KUKA KRL program: ps_601s1.src, ps_601s1.dat

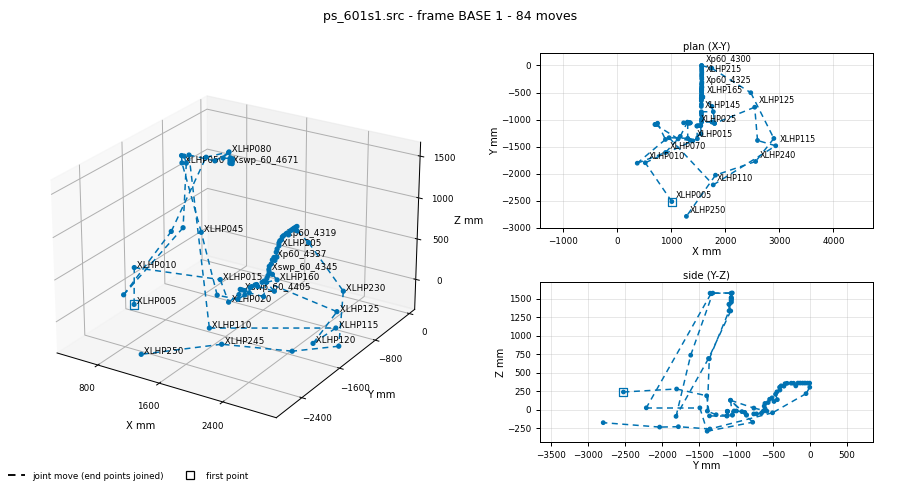
[picture p0: tool path of ps_601s1.src in frame BASE 1, 84 of 89 moves have a stored position in this frame; points joined in program order, loops and branches not executed]
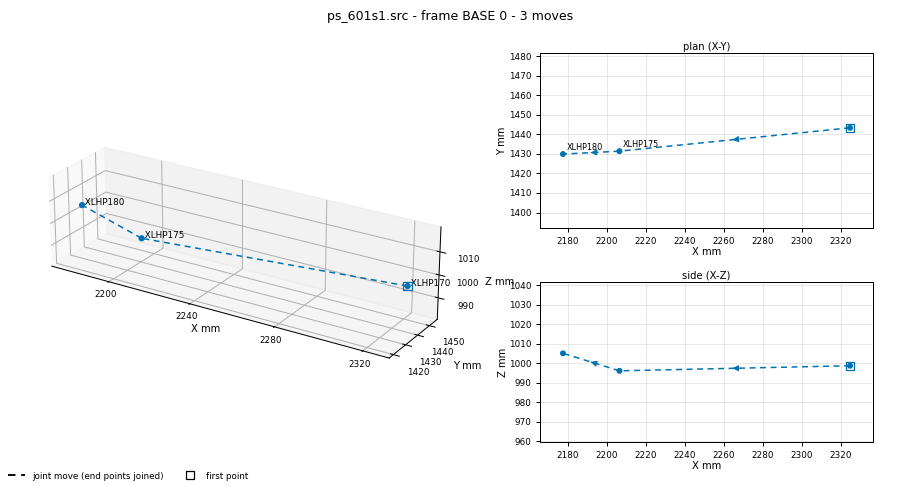
[picture p1: tool path of ps_601s1.src in frame BASE 0, 3 of 89 moves have a stored position in this frame; points joined in program order, loops and branches not executed]
--- ps_601s1.src ---
&ACCESS RVO2
&REL 23
&COMMENT Solda Respot C1 STB
DEF ps_601s1( )
EXT e_Fraes_1()
EXT f_Fraes_1()
;FOLD INI
   ;FOLD BASISTECH INI
      GLOBAL INTERRUPT DECL 3 WHEN $STOPMESS==TRUE DO IR_STOPM ( )
      INTERRUPT ON 3
      BAS (#INITMOV,0 )
   ;ENDFOLD (BASISTECH INI)
   ;FOLD SPOTTECH INI
      USERSPOT(#INIT)
   ;ENDFOLD (SPOTTECH INI)
   ;FOLD GRIPPERTECH INI
      USER_GRP(0,DUMMY,DUMMY,GDEFAULT)
   ;ENDFOLD (GRIPPERTECH INI)
   ;FOLD USER INI
      ;Make your modifications here

   ;ENDFOLD (USER INI)
;ENDFOLD (INI)

; Estacao P13.060 - Robo R1
; Programa: Solda Respot C1 (STB)
; Caracterização dos meios de produção:
; 02/09/2014 09:15 Changes by KUKA Roboter do Brasil

chk_w1_wechs_ok ( )           ; CHECK FERRAMENTA: C1

;FOLD PTP HOME  Vel= 70 % DEFAULT;%{PE}%R 4.1.16,%MKUKATPBASIS,%CMOVE,%VPTP,%P 1:PTP, 2:HOME, 3:, 5:70, 7:DEFAULT
$BWDSTART = FALSE
PDAT_ACT=PDEFAULT
BAS(#PTP_DAT)
FDAT_ACT=FHOME
BAS(#FRAMES)
BAS(#VEL_PTP,70)
$H_POS=XHOME
PTP XHOME
;ENDFOLD

IF (NOT(GHOST())) THEN
IF MaxStandMenge (1) THEN
  MaxStandmengeErreicht (1)
ENDIF

IF Elektrodenwechsel (1) THEN
  e_Fraes_1()
ENDIF
ENDIF

;FOLD OUT 3364 'R1_Solicita Lib. Soldar Geo2' State=TRUE ;%{PE}%R 8.2.20,%MKUKATPBASIS,%COUT,%VOUTX,%P 2:3364, 3:R1_Solicita Lib. Soldar Geo2, 5:TRUE, 6:
$OUT[3364]=TRUE
;ENDFOLD
;FOLD WAIT FOR ( IN 3334 'R1_Aguarda Lib. Soldar Respot' );%{PE}%R 8.2.20,%MKUKATPBASIS,%CEXT_WAIT_FOR,%VEXT_WAIT_FOR,%P 2:, 4:, 5:$IN, 6:3334, 7:R1_Aguarda Lib. Soldar Respot, 9:
WAIT FOR  ( $IN[3334] )
;ENDFOLD
;FOLD OUT 3364 'R1_Solicita Lib. Soldar Geo2' State=FALSE ;%{PE}%R 8.2.20,%MKUKATPBASIS,%COUT,%VOUTX,%P 2:3364, 3:R1_Solicita Lib. Soldar Geo2, 5:FALSE, 6:
$OUT[3364]=FALSE
;ENDFOLD

;FOLD PTP LHP005 CONT Vel=70 % P_OLP1 Tool[1] Base[1];%{PE}%R 4.1.15,%MKUKATPBASIS,%CMOVE,%VPTP,%P 1:PTP, 2:LHP005, 3:C_PTP, 5:70, 7:P_OLP1
$BWDSTART=FALSE
PDAT_ACT=PP_OLP1
BAS (#PTP_DAT )
FDAT_ACT=FLHP005
BAS (#FRAMES )
BAS (#VEL_PTP,70 )
PTP  XLHP005 C_PTP
;ENDFOLD
;FOLD PTP LHP010 CONT Vel= 70 % P_OLP2 Tool[1]:GUN C1 Base[1]:Actros ;%{PE}%R 4.1.16,%MKUKATPBASIS,%CMOVE,%VPTP,%P 1:PTP, 2:LHP010, 3:C_PTP, 5:70, 7:P_OLP2
$BWDSTART = FALSE
PDAT_ACT=PP_OLP2
BAS(#PTP_DAT)
FDAT_ACT=FLHP010
BAS(#FRAMES)
BAS(#VEL_PTP,70)
PTP XLHP010 C_PTP
;ENDFOLD
;FOLD PTP LHP015 CONT Vel= 60 % P_OLP3 Tool[1]:GUN C1 Base[1]:Actros ;%{PE}%R 4.1.16,%MKUKATPBASIS,%CMOVE,%VPTP,%P 1:PTP, 2:LHP015, 3:C_PTP, 5:60, 7:P_OLP3
$BWDSTART = FALSE
PDAT_ACT=PP_OLP3
BAS(#PTP_DAT)
FDAT_ACT=FLHP015
BAS(#FRAMES)
BAS(#VEL_PTP,60)
PTP XLHP015 C_PTP
;ENDFOLD
;FOLD PTP LHP020 CONT Vel= 50 % P_OLP4 Tool[1]:GUN C1 Base[1]:Actros ;%{PE}%R 4.1.16,%MKUKATPBASIS,%CMOVE,%VPTP,%P 1:PTP, 2:LHP020, 3:C_PTP, 5:50, 7:P_OLP4
$BWDSTART = FALSE
PDAT_ACT=PP_OLP4
BAS(#PTP_DAT)
FDAT_ACT=FLHP020
BAS(#FRAMES)
BAS(#VEL_PTP,50)
PTP XLHP020 C_PTP
;ENDFOLD

;FOLD OUT 3331 'R1_Soldando' State=TRUE ;%{PE}%R 8.2.20,%MKUKATPBASIS,%COUT,%VOUTX,%P 2:3331, 3:R1_Soldando, 5:TRUE, 6:
$OUT[3331]=TRUE
;ENDFOLD
;FOLD OUT 3369 'Area de Solda' State=FALSE ;%{PE}%R 8.2.20,%MKUKATPBASIS,%COUT,%VOUTX,%P 2:3369, 3:Area de Solda, 5:FALSE, 6:
$OUT[3369]=FALSE
;ENDFOLD

; Retract Close
;FOLD PTP LHP025 PDAT1 RETR CLS Gun= 1 Tool[1]:GUN C1 Base[1]:Actros ;%{PE}%R 4.1.12,%MKUKATPSPOT,%CRETR,%VPTP,%P 1:PTP, 2:LHP025, 3:, 5:100, 7:PDAT1, 9:#CLO, 11:1, 13:#FIRST
$BWDSTART = TRUE
PDAT_ACT=PPDAT1
BAS(#PTP_DAT)
FDAT_ACT=FLHP025
BAS(#FRAMES)
BAS(#VEL_PTP,PPDAT1.VEL)
S_ACT.GUN=1
S_ACT.PAIR=#FIRST
S_ACT.RETR=#CLO
S_READY=FALSE
PTP XLHP025
USERSPOT(#RETR, S_ACT)
WAIT FOR S_READY
;ENDFOLD

;FOLD ; SWP_60_4413;%{PE}%R2.2,%MKUKATPBASIS,%CCOMMENT,%VNORMAL,%P 2: SWP_60_4413
;ENDFOLD
;FOLD PTP swp_60_4413 PDAT3 SPOT Gun= 1 RETR CLS PgNo1= 106 ACTIVE= 1 Tool[1]:GUN C1 Base[1]:Actros ;%{PE}%R 4.1.12,%MKUKATPSPOT,%CSPOT,%VPTP,%P 1:PTP, 2:swp_60_4413, 3:, 5:100, 7:PDAT3, 10:1, 12:#FIRST, 14:#CLO, 16:106, 18:1, 20:0, 22:0, 24:1, 25:NORMAL
$BWDSTART = TRUE
PDAT_ACT=PPDAT3
BAS(#PTP_DAT)
FDAT_ACT=Fswp_60_4413
BAS(#FRAMES)
BAS(#VEL_PTP,PPDAT3.VEL)
S_ACT.GUN=1
S_ACT.PAIR=SDEFAULT.PAIR
S_ACT.RETR=#CLO
S_ACT.CLO_TM=1
S_ACT.PGNO1=106
S_ACT.PGNO2=SDEFAULT.PGNO2
S_ACT.PRESS1=SDEFAULT.PRESS1
S_ACT.PRESS2=SDEFAULT.PRESS2
S_READY=FALSE
PTP Xswp_60_4413
USERSPOT(#SPOT, S_ACT)
WAIT FOR S_READY
;ENDFOLD

;FOLD ; SWP_60_4405;%{PE}%R2.2,%MKUKATPBASIS,%CCOMMENT,%VNORMAL,%P 2: SWP_60_4405
;ENDFOLD
;FOLD PTP swp_60_4405 PDAT4 SPOT Gun= 1 RETR CLS PgNo1= 107 ACTIVE= 1 Tool[1]:GUN C1 Base[1]:Actros ;%{PE}%R 4.1.12,%MKUKATPSPOT,%CSPOT,%VPTP,%P 1:PTP, 2:swp_60_4405, 3:, 5:100, 7:PDAT4, 10:1, 12:#FIRST, 14:#CLO, 16:107, 18:1, 20:0, 22:0, 24:1, 25:NORMAL
$BWDSTART = TRUE
PDAT_ACT=PPDAT4
BAS(#PTP_DAT)
FDAT_ACT=Fswp_60_4405
BAS(#FRAMES)
BAS(#VEL_PTP,PPDAT4.VEL)
S_ACT.GUN=1
S_ACT.PAIR=SDEFAULT.PAIR
S_ACT.RETR=#CLO
S_ACT.CLO_TM=1
S_ACT.PGNO1=107
S_ACT.PGNO2=SDEFAULT.PGNO2
S_ACT.PRESS1=SDEFAULT.PRESS1
S_ACT.PRESS2=SDEFAULT.PRESS2
S_READY=FALSE
PTP Xswp_60_4405
USERSPOT(#SPOT, S_ACT)
WAIT FOR S_READY
;ENDFOLD

;FOLD ; SWP_60_4409;%{PE}%R2.2,%MKUKATPBASIS,%CCOMMENT,%VNORMAL,%P 2: SWP_60_4409
;ENDFOLD
;FOLD PTP swp_60_4409 PDAT5 SPOT Gun= 1 RETR CLS PgNo1= 108 ACTIVE= 1 Tool[1]:GUN C1 Base[1]:Actros ;%{PE}%R 4.1.12,%MKUKATPSPOT,%CSPOT,%VPTP,%P 1:PTP, 2:swp_60_4409, 3:, 5:100, 7:PDAT5, 10:1, 12:#FIRST, 14:#CLO, 16:108, 18:1, 20:0, 22:0, 24:1, 25:NORMAL
$BWDSTART = TRUE
PDAT_ACT=PPDAT5
BAS(#PTP_DAT)
FDAT_ACT=Fswp_60_4409
BAS(#FRAMES)
BAS(#VEL_PTP,PPDAT5.VEL)
S_ACT.GUN=1
S_ACT.PAIR=SDEFAULT.PAIR
S_ACT.RETR=#CLO
S_ACT.CLO_TM=1
S_ACT.PGNO1=108
S_ACT.PGNO2=SDEFAULT.PGNO2
S_ACT.PRESS1=SDEFAULT.PRESS1
S_ACT.PRESS2=SDEFAULT.PRESS2
S_READY=FALSE
PTP Xswp_60_4409
USERSPOT(#SPOT, S_ACT)
WAIT FOR S_READY
;ENDFOLD

;FOLD PTP LHP030 PDAT78 RETR OPN Gun= 1 Tool[1]:GUN C1 Base[1]:Actros ;%{PE}%R 4.1.12,%MKUKATPSPOT,%CRETR,%VPTP,%P 1:PTP, 2:LHP030, 3:, 5:100, 7:PDAT78, 9:#OPN, 11:1, 13:#FIRST
$BWDSTART = TRUE
PDAT_ACT=PPDAT78
BAS(#PTP_DAT)
FDAT_ACT=FLHP030
BAS(#FRAMES)
BAS(#VEL_PTP,PPDAT78.VEL)
S_ACT.GUN=1
S_ACT.PAIR=#FIRST
S_ACT.RETR=#OPN
S_READY=FALSE
PTP XLHP030
USERSPOT(#RETR, S_ACT)
WAIT FOR S_READY
;ENDFOLD
;FOLD PTP LHP035 CONT Vel= 50 % P_OLP10 Tool[1]:GUN C1 Base[1]:Actros ;%{PE}%R 4.1.16,%MKUKATPBASIS,%CMOVE,%VPTP,%P 1:PTP, 2:LHP035, 3:C_PTP, 5:50, 7:P_OLP10
$BWDSTART = FALSE
PDAT_ACT=PP_OLP10
BAS(#PTP_DAT)
FDAT_ACT=FLHP035
BAS(#FRAMES)
BAS(#VEL_PTP,50)
PTP XLHP035 C_PTP
;ENDFOLD
;FOLD PTP LHP040 CONT Vel= 65 % PDAT68 Tool[1]:GUN C1 Base[1]:Actros ;%{PE}%R 4.1.16,%MKUKATPBASIS,%CMOVE,%VPTP,%P 1:PTP, 2:LHP040, 3:C_PTP, 5:65, 7:PDAT68
$BWDSTART = FALSE
PDAT_ACT=PPDAT68
BAS(#PTP_DAT)
FDAT_ACT=FLHP040
BAS(#FRAMES)
BAS(#VEL_PTP,65)
PTP XLHP040 C_PTP
;ENDFOLD

;FOLD ; PONTOS INSERIDOS DO ROBO 3;%{PE}%R 4.1.16,%MKUKATPBASIS,%CCOMMENT,%VNORMAL,%P 2:PONTOS INSERIDOS DO ROBO 3
;ENDFOLD

;FOLD PTP LHP045 CONT Vel= 65 % PDAT72 Tool[1]:GUN C1 Base[1]:Actros ;%{PE}%R 4.1.16,%MKUKATPBASIS,%CMOVE,%VPTP,%P 1:PTP, 2:LHP045, 3:C_PTP, 5:65, 7:PDAT72
$BWDSTART = FALSE
PDAT_ACT=PPDAT72
BAS(#PTP_DAT)
FDAT_ACT=FLHP045
BAS(#FRAMES)
BAS(#VEL_PTP,65)
PTP XLHP045 C_PTP
;ENDFOLD
;FOLD PTP LHP050 CONT Vel= 70 % PDAT93 Tool[1]:GUN C1 Base[1]:Actros ;%{PE}%R 4.1.16,%MKUKATPBASIS,%CMOVE,%VPTP,%P 1:PTP, 2:LHP050, 3:C_PTP, 5:70, 7:PDAT93
$BWDSTART = FALSE
PDAT_ACT=PPDAT93
BAS(#PTP_DAT)
FDAT_ACT=FLHP050
BAS(#FRAMES)
BAS(#VEL_PTP,70)
PTP XLHP050 C_PTP
;ENDFOLD

;FOLD ; SWP_60_5627;%{PE}%R 4.1.16,%MKUKATPBASIS,%CCOMMENT,%VNORMAL,%P 2:SWP_60_5627
;ENDFOLD
;FOLD PTP SWP_60_5627 PDAT74 SPOT Gun= 1 RETR CLS PgNo1= 109 ACTIVE= 1 Tool[1]:GUN C1 Base[1]:Actros ;%{PE}%R 4.1.12,%MKUKATPSPOT,%CSPOT,%VPTP,%P 1:PTP, 2:SWP_60_5627, 3:, 5:100, 7:PDAT74, 10:1, 12:#FIRST, 14:#CLO, 16:109, 18:1, 20:0, 22:0, 24:1, 25:NORMAL
$BWDSTART = TRUE
PDAT_ACT=PPDAT74
BAS(#PTP_DAT)
FDAT_ACT=FSWP_60_5627
BAS(#FRAMES)
BAS(#VEL_PTP,PPDAT74.VEL)
S_ACT.GUN=1
S_ACT.PAIR=SDEFAULT.PAIR
S_ACT.RETR=#CLO
S_ACT.CLO_TM=1
S_ACT.PGNO1=109
S_ACT.PGNO2=SDEFAULT.PGNO2
S_ACT.PRESS1=SDEFAULT.PRESS1
S_ACT.PRESS2=SDEFAULT.PRESS2
S_READY=FALSE
PTP XSWP_60_5627
USERSPOT(#SPOT, S_ACT)
WAIT FOR S_READY
;ENDFOLD

;FOLD ; SWP_60_5633;%{PE}%R 4.1.16,%MKUKATPBASIS,%CCOMMENT,%VNORMAL,%P 2:SWP_60_5633
;ENDFOLD
;FOLD PTP SWP_60_5633 PDAT75 SPOT Gun= 1 RETR OPN PgNo1= 110 ACTIVE= 1 Tool[1]:GUN C1 Base[1]:Actros ;%{PE}%R 4.1.12,%MKUKATPSPOT,%CSPOT,%VPTP,%P 1:PTP, 2:SWP_60_5633, 3:, 5:100, 7:PDAT75, 10:1, 12:#FIRST, 14:#OPN, 16:110, 18:1, 20:0, 22:0, 24:1, 25:NORMAL
$BWDSTART = TRUE
PDAT_ACT=PPDAT75
BAS(#PTP_DAT)
FDAT_ACT=FSWP_60_5633
BAS(#FRAMES)
BAS(#VEL_PTP,PPDAT75.VEL)
S_ACT.GUN=1
S_ACT.PAIR=SDEFAULT.PAIR
S_ACT.RETR=#OPN
S_ACT.CLO_TM=1
S_ACT.PGNO1=110
S_ACT.PGNO2=SDEFAULT.PGNO2
S_ACT.PRESS1=SDEFAULT.PRESS1
S_ACT.PRESS2=SDEFAULT.PRESS2
S_READY=FALSE
PTP XSWP_60_5633
USERSPOT(#SPOT, S_ACT)
WAIT FOR S_READY
;ENDFOLD

;FOLD PTP LHP055 CONT Vel= 55 % PDAT76 Tool[1]:GUN C1 Base[1]:Actros ;%{PE}%R 4.1.16,%MKUKATPBASIS,%CMOVE,%VPTP,%P 1:PTP, 2:LHP055, 3:C_PTP, 5:55, 7:PDAT76
$BWDSTART = FALSE
PDAT_ACT=PPDAT76
BAS(#PTP_DAT)
FDAT_ACT=FLHP055
BAS(#FRAMES)
BAS(#VEL_PTP,55)
PTP XLHP055 C_PTP
;ENDFOLD

;FOLD ; FIM DOS PONTOS INSERIDOS;%{PE}%R 4.1.16,%MKUKATPBASIS,%CCOMMENT,%VNORMAL,%P 2:FIM DOS PONTOS INSERIDOS
;ENDFOLD

;FOLD PTP LHP060 CONT Vel= 65 % PDAT7 Tool[1]:GUN C1 Base[1]:Actros ;%{PE}%R 4.1.16,%MKUKATPBASIS,%CMOVE,%VPTP,%P 1:PTP, 2:LHP060, 3:C_PTP, 5:65, 7:PDAT7
$BWDSTART = FALSE
PDAT_ACT=PPDAT7
BAS(#PTP_DAT)
FDAT_ACT=FLHP060
BAS(#FRAMES)
BAS(#VEL_PTP,65)
PTP XLHP060 C_PTP
;ENDFOLD
;FOLD PTP LHP065 CONT Vel= 70 % PDAT8 Tool[1]:GUN C1 Base[1]:Actros ;%{PE}%R 4.1.16,%MKUKATPBASIS,%CMOVE,%VPTP,%P 1:PTP, 2:LHP065, 3:C_PTP, 5:70, 7:PDAT8
$BWDSTART = FALSE
PDAT_ACT=PPDAT8
BAS(#PTP_DAT)
FDAT_ACT=FLHP065
BAS(#FRAMES)
BAS(#VEL_PTP,70)
PTP XLHP065 C_PTP
;ENDFOLD
;FOLD PTP LHP070 CONT Vel= 70 % P_OLP12 Tool[1]:GUN C1 Base[1]:Actros ;%{PE}%R 4.1.16,%MKUKATPBASIS,%CMOVE,%VPTP,%P 1:PTP, 2:LHP070, 3:C_PTP, 5:70, 7:P_OLP12
$BWDSTART = FALSE
PDAT_ACT=PP_OLP12
BAS(#PTP_DAT)
FDAT_ACT=FLHP070
BAS(#FRAMES)
BAS(#VEL_PTP,70)
PTP XLHP070 C_PTP
;ENDFOLD
;FOLD PTP LHP075 CONT Vel= 70 % P_OLP13 Tool[1]:GUN C1 Base[1]:Actros ;%{PE}%R 4.1.16,%MKUKATPBASIS,%CMOVE,%VPTP,%P 1:PTP, 2:LHP075, 3:C_PTP, 5:70, 7:P_OLP13
$BWDSTART = FALSE
PDAT_ACT=PP_OLP13
BAS(#PTP_DAT)
FDAT_ACT=FLHP075
BAS(#FRAMES)
BAS(#VEL_PTP,70)
PTP XLHP075 C_PTP
;ENDFOLD
;FOLD PTP LHP080 PDAT9 RETR OPN Gun= 1 Tool[1]:GUN C1 Base[1]:Actros ;%{PE}%R 4.1.12,%MKUKATPSPOT,%CRETR,%VPTP,%P 1:PTP, 2:LHP080, 3:, 5:100, 7:PDAT9, 9:#OPN, 11:1, 13:#FIRST
$BWDSTART = TRUE
PDAT_ACT=PPDAT9
BAS(#PTP_DAT)
FDAT_ACT=FLHP080
BAS(#FRAMES)
BAS(#VEL_PTP,PPDAT9.VEL)
S_ACT.GUN=1
S_ACT.PAIR=#FIRST
S_ACT.RETR=#OPN
S_READY=FALSE
PTP XLHP080
USERSPOT(#RETR, S_ACT)
WAIT FOR S_READY
;ENDFOLD
;FOLD PTP LHP085 PDAT10 RETR CLS Gun= 1 Tool[1]:GUN C1 Base[1]:Actros ;%{PE}%R 4.1.12,%MKUKATPSPOT,%CRETR,%VPTP,%P 1:PTP, 2:LHP085, 3:, 5:100, 7:PDAT10, 9:#CLO, 11:1, 13:#FIRST
$BWDSTART = TRUE
PDAT_ACT=PPDAT10
BAS(#PTP_DAT)
FDAT_ACT=FLHP085
BAS(#FRAMES)
BAS(#VEL_PTP,PPDAT10.VEL)
S_ACT.GUN=1
S_ACT.PAIR=#FIRST
S_ACT.RETR=#CLO
S_READY=FALSE
PTP XLHP085
USERSPOT(#RETR, S_ACT)
WAIT FOR S_READY
;ENDFOLD

;FOLD ; SWP_60_4663;%{PE}%R2.2,%MKUKATPBASIS,%CCOMMENT,%VNORMAL,%P 2: SWP_60_4663
;ENDFOLD
;FOLD PTP swp_60_4663 PDAT11 SPOT Gun= 1 RETR CLS PgNo1= 111 ACTIVE= 1 Tool[1]:GUN C1 Base[1]:Actros ;%{PE}%R 4.1.12,%MKUKATPSPOT,%CSPOT,%VPTP,%P 1:PTP, 2:swp_60_4663, 3:, 5:100, 7:PDAT11, 10:1, 12:#FIRST, 14:#CLO, 16:111, 18:1, 20:0, 22:0, 24:1, 25:NORMAL
$BWDSTART = TRUE
PDAT_ACT=PPDAT11
BAS(#PTP_DAT)
FDAT_ACT=Fswp_60_4663
BAS(#FRAMES)
BAS(#VEL_PTP,PPDAT11.VEL)
S_ACT.GUN=1
S_ACT.PAIR=SDEFAULT.PAIR
S_ACT.RETR=#CLO
S_ACT.CLO_TM=1
S_ACT.PGNO1=111
S_ACT.PGNO2=SDEFAULT.PGNO2
S_ACT.PRESS1=SDEFAULT.PRESS1
S_ACT.PRESS2=SDEFAULT.PRESS2
S_READY=FALSE
PTP Xswp_60_4663
USERSPOT(#SPOT, S_ACT)
WAIT FOR S_READY
;ENDFOLD

;FOLD ; SWP_60_4667;%{PE}%R2.2,%MKUKATPBASIS,%CCOMMENT,%VNORMAL,%P 2: SWP_60_4667
;ENDFOLD
;FOLD PTP swp_60_4667 PDAT12 SPOT Gun= 1 RETR CLS PgNo1= 112 ACTIVE= 1 Tool[1]:GUN C1 Base[1]:Actros ;%{PE}%R 4.1.12,%MKUKATPSPOT,%CSPOT,%VPTP,%P 1:PTP, 2:swp_60_4667, 3:, 5:100, 7:PDAT12, 10:1, 12:#FIRST, 14:#CLO, 16:112, 18:1, 20:0, 22:0, 24:1, 25:NORMAL
$BWDSTART = TRUE
PDAT_ACT=PPDAT12
BAS(#PTP_DAT)
FDAT_ACT=Fswp_60_4667
BAS(#FRAMES)
BAS(#VEL_PTP,PPDAT12.VEL)
S_ACT.GUN=1
S_ACT.PAIR=SDEFAULT.PAIR
S_ACT.RETR=#CLO
S_ACT.CLO_TM=1
S_ACT.PGNO1=112
S_ACT.PGNO2=SDEFAULT.PGNO2
S_ACT.PRESS1=SDEFAULT.PRESS1
S_ACT.PRESS2=SDEFAULT.PRESS2
S_READY=FALSE
PTP Xswp_60_4667
USERSPOT(#SPOT, S_ACT)
WAIT FOR S_READY
;ENDFOLD

;FOLD ; SWP_60_4671;%{PE}%R2.2,%MKUKATPBASIS,%CCOMMENT,%VNORMAL,%P 2: SWP_60_4671
;ENDFOLD
;FOLD PTP swp_60_4671 PDAT14 SPOT Gun= 1 RETR CLS PgNo1= 113 ACTIVE= 1 Tool[1]:GUN C1 Base[1]:Actros ;%{PE}%R 4.1.12,%MKUKATPSPOT,%CSPOT,%VPTP,%P 1:PTP, 2:swp_60_4671, 3:, 5:100, 7:PDAT14, 10:1, 12:#FIRST, 14:#CLO, 16:113, 18:1, 20:0, 22:0, 24:1, 25:NORMAL
$BWDSTART = TRUE
PDAT_ACT=PPDAT14
BAS(#PTP_DAT)
FDAT_ACT=Fswp_60_4671
BAS(#FRAMES)
BAS(#VEL_PTP,PPDAT14.VEL)
S_ACT.GUN=1
S_ACT.PAIR=SDEFAULT.PAIR
S_ACT.RETR=#CLO
S_ACT.CLO_TM=1
S_ACT.PGNO1=113
S_ACT.PGNO2=SDEFAULT.PGNO2
S_ACT.PRESS1=SDEFAULT.PRESS1
S_ACT.PRESS2=SDEFAULT.PRESS2
S_READY=FALSE
PTP Xswp_60_4671
USERSPOT(#SPOT, S_ACT)
WAIT FOR S_READY
;ENDFOLD

;FOLD ; SWP_60_4675;%{PE}%R2.2,%MKUKATPBASIS,%CCOMMENT,%VNORMAL,%P 2: SWP_60_4675
;ENDFOLD
;FOLD PTP swp_60_4675 PDAT15 SPOT Gun= 1 RETR CLS PgNo1= 114 ACTIVE= 1 Tool[1]:GUN C1 Base[1]:Actros ;%{PE}%R 4.1.12,%MKUKATPSPOT,%CSPOT,%VPTP,%P 1:PTP, 2:swp_60_4675, 3:, 5:100, 7:PDAT15, 10:1, 12:#FIRST, 14:#CLO, 16:114, 18:1, 20:0, 22:0, 24:1, 25:NORMAL
$BWDSTART = TRUE
PDAT_ACT=PPDAT15
BAS(#PTP_DAT)
FDAT_ACT=Fswp_60_4675
BAS(#FRAMES)
BAS(#VEL_PTP,PPDAT15.VEL)
S_ACT.GUN=1
S_ACT.PAIR=SDEFAULT.PAIR
S_ACT.RETR=#CLO
S_ACT.CLO_TM=1
S_ACT.PGNO1=114
S_ACT.PGNO2=SDEFAULT.PGNO2
S_ACT.PRESS1=SDEFAULT.PRESS1
S_ACT.PRESS2=SDEFAULT.PRESS2
S_READY=FALSE
PTP Xswp_60_4675
USERSPOT(#SPOT, S_ACT)
WAIT FOR S_READY
;ENDFOLD

;FOLD ; SWP_60_4669;%{PE}%R2.2,%MKUKATPBASIS,%CCOMMENT,%VNORMAL,%P 2: SWP_60_4669
;ENDFOLD
;FOLD PTP swp_60_4669 PDAT16 SPOT Gun= 1 RETR CLS PgNo1= 115 ACTIVE= 1 Tool[1]:GUN C1 Base[1]:Actros ;%{PE}%R 4.1.12,%MKUKATPSPOT,%CSPOT,%VPTP,%P 1:PTP, 2:swp_60_4669, 3:, 5:100, 7:PDAT16, 10:1, 12:#FIRST, 14:#CLO, 16:115, 18:1, 20:0, 22:0, 24:1, 25:NORMAL
$BWDSTART = TRUE
PDAT_ACT=PPDAT16
BAS(#PTP_DAT)
FDAT_ACT=Fswp_60_4669
BAS(#FRAMES)
BAS(#VEL_PTP,PPDAT16.VEL)
S_ACT.GUN=1
S_ACT.PAIR=SDEFAULT.PAIR
S_ACT.RETR=#CLO
S_ACT.CLO_TM=1
S_ACT.PGNO1=115
S_ACT.PGNO2=SDEFAULT.PGNO2
S_ACT.PRESS1=SDEFAULT.PRESS1
S_ACT.PRESS2=SDEFAULT.PRESS2
S_READY=FALSE
PTP Xswp_60_4669
USERSPOT(#SPOT, S_ACT)
WAIT FOR S_READY
;ENDFOLD

;FOLD ; SWP_60_4665;%{PE}%R2.2,%MKUKATPBASIS,%CCOMMENT,%VNORMAL,%P 2: SWP_60_4665
;ENDFOLD
;FOLD PTP swp_60_4665 PDAT13 SPOT Gun= 1 RETR CLS PgNo1= 116 ACTIVE= 1 Tool[1]:GUN C1 Base[1]:Actros ;%{PE}%R 4.1.12,%MKUKATPSPOT,%CSPOT,%VPTP,%P 1:PTP, 2:swp_60_4665, 3:, 5:100, 7:PDAT13, 10:1, 12:#FIRST, 14:#CLO, 16:116, 18:1, 20:0, 22:0, 24:1, 25:NORMAL
$BWDSTART = TRUE
PDAT_ACT=PPDAT13
BAS(#PTP_DAT)
FDAT_ACT=Fswp_60_4665
BAS(#FRAMES)
BAS(#VEL_PTP,PPDAT13.VEL)
S_ACT.GUN=1
S_ACT.PAIR=SDEFAULT.PAIR
S_ACT.RETR=#CLO
S_ACT.CLO_TM=1
S_ACT.PGNO1=116
S_ACT.PGNO2=SDEFAULT.PGNO2
S_ACT.PRESS1=SDEFAULT.PRESS1
S_ACT.PRESS2=SDEFAULT.PRESS2
S_READY=FALSE
PTP Xswp_60_4665
USERSPOT(#SPOT, S_ACT)
WAIT FOR S_READY
;ENDFOLD

;FOLD PTP LHP090 PDAT17 RETR OPN Gun= 1 Tool[1]:GUN C1 Base[1]:Actros ;%{PE}%R 4.1.12,%MKUKATPSPOT,%CRETR,%VPTP,%P 1:PTP, 2:LHP090, 3:, 5:100, 7:PDAT17, 9:#OPN, 11:1, 13:#FIRST
$BWDSTART = TRUE
PDAT_ACT=PPDAT17
BAS(#PTP_DAT)
FDAT_ACT=FLHP090
BAS(#FRAMES)
BAS(#VEL_PTP,PPDAT17.VEL)
S_ACT.GUN=1
S_ACT.PAIR=#FIRST
S_ACT.RETR=#OPN
S_READY=FALSE
PTP XLHP090
USERSPOT(#RETR, S_ACT)
WAIT FOR S_READY
;ENDFOLD
;FOLD PTP LHP095  Vel= 60 % P_OLP22 Tool[1]:GUN C1 Base[1]:Actros ;%{PE}%R 4.1.16,%MKUKATPBASIS,%CMOVE,%VPTP,%P 1:PTP, 2:LHP095, 3:, 5:60, 7:P_OLP22
$BWDSTART = FALSE
PDAT_ACT=PP_OLP22
BAS(#PTP_DAT)
FDAT_ACT=FLHP095
BAS(#FRAMES)
BAS(#VEL_PTP,60)
PTP XLHP095
;ENDFOLD
;FOLD PTP LHP100 CONT Vel= 70 % P_OLP23 Tool[1]:GUN C1 Base[1]:Actros ;%{PE}%R 4.1.16,%MKUKATPBASIS,%CMOVE,%VPTP,%P 1:PTP, 2:LHP100, 3:C_PTP, 5:70, 7:P_OLP23
$BWDSTART = FALSE
PDAT_ACT=PP_OLP23
BAS(#PTP_DAT)
FDAT_ACT=FLHP100
BAS(#FRAMES)
BAS(#VEL_PTP,70)
PTP XLHP100 C_PTP
;ENDFOLD
;FOLD PTP LHP105  Vel= 70 % P_OLP24 Tool[1]:GUN C1 Base[1]:Actros ;%{PE}%R 4.1.16,%MKUKATPBASIS,%CMOVE,%VPTP,%P 1:PTP, 2:LHP105, 3:, 5:70, 7:P_OLP24
$BWDSTART = FALSE
PDAT_ACT=PP_OLP24
BAS(#PTP_DAT)
FDAT_ACT=FLHP105
BAS(#FRAMES)
BAS(#VEL_PTP,70)
PTP XLHP105
;ENDFOLD
;FOLD PTP LHP110 CONT Vel= 70 % P_OLP25 Tool[1]:GUN C1 Base[1]:Actros ;%{PE}%R 4.1.16,%MKUKATPBASIS,%CMOVE,%VPTP,%P 1:PTP, 2:LHP110, 3:C_PTP, 5:70, 7:P_OLP25
$BWDSTART = FALSE
PDAT_ACT=PP_OLP25
BAS(#PTP_DAT)
FDAT_ACT=FLHP110
BAS(#FRAMES)
BAS(#VEL_PTP,70)
PTP XLHP110 C_PTP
;ENDFOLD
;FOLD PTP LHP115 CONT Vel= 65 % P_OLP26 Tool[1]:GUN C1 Base[1]:Actros ;%{PE}%R 4.1.16,%MKUKATPBASIS,%CMOVE,%VPTP,%P 1:PTP, 2:LHP115, 3:C_PTP, 5:65, 7:P_OLP26
$BWDSTART = FALSE
PDAT_ACT=PP_OLP26
BAS(#PTP_DAT)
FDAT_ACT=FLHP115
BAS(#FRAMES)
BAS(#VEL_PTP,65)
PTP XLHP115 C_PTP
;ENDFOLD
;FOLD PTP LHP120 CONT Vel= 60 % PDAT77 Tool[1]:GUN C1 Base[1]:Actros ;%{PE}%R 4.1.16,%MKUKATPBASIS,%CMOVE,%VPTP,%P 1:PTP, 2:LHP120, 3:C_PTP, 5:60, 7:PDAT77
$BWDSTART = FALSE
PDAT_ACT=PPDAT77
BAS(#PTP_DAT)
FDAT_ACT=FLHP120
BAS(#FRAMES)
BAS(#VEL_PTP,60)
PTP XLHP120 C_PTP
;ENDFOLD

;FOLD ; start interlock R2;%{PE}%R 4.1.16,%MKUKATPBASIS,%CCOMMENT,%VNORMAL,%P 2:start interlock R2
;ENDFOLD
;FOLD Kollision.Ueberwachung_2_Ein ;%{PE}%MKUKATPUSER
COLLSTOP( 2, 1 ) ;INTERRUPTUEBERWACHT
;ENDFOLD

;FOLD PTP LHP125 CONT Vel= 60 % P_OLP27 Tool[1]:GUN C1 Base[1]:Actros ;%{PE}%R 4.1.16,%MKUKATPBASIS,%CMOVE,%VPTP,%P 1:PTP, 2:LHP125, 3:C_PTP, 5:60, 7:P_OLP27
$BWDSTART = FALSE
PDAT_ACT=PP_OLP27
BAS(#PTP_DAT)
FDAT_ACT=FLHP125
BAS(#FRAMES)
BAS(#VEL_PTP,60)
PTP XLHP125 C_PTP
;ENDFOLD
;FOLD PTP LHP130 CONT Vel= 60 % P_OLP28 Tool[1]:GUN C1 Base[1]:Actros ;%{PE}%R 4.1.16,%MKUKATPBASIS,%CMOVE,%VPTP,%P 1:PTP, 2:LHP130, 3:C_PTP, 5:60, 7:P_OLP28
$BWDSTART = FALSE
PDAT_ACT=PP_OLP28
BAS(#PTP_DAT)
FDAT_ACT=FLHP130
BAS(#FRAMES)
BAS(#VEL_PTP,60)
PTP XLHP130 C_PTP
;ENDFOLD
;FOLD PTP LHP135 CONT Vel= 55 % P_OLP29 Tool[1]:GUN C1 Base[1]:Actros ;%{PE}%R 4.1.16,%MKUKATPBASIS,%CMOVE,%VPTP,%P 1:PTP, 2:LHP135, 3:C_PTP, 5:55, 7:P_OLP29
$BWDSTART = FALSE
PDAT_ACT=PP_OLP29
BAS(#PTP_DAT)
FDAT_ACT=FLHP135
BAS(#FRAMES)
BAS(#VEL_PTP,55)
PTP XLHP135 C_PTP
;ENDFOLD
;FOLD PTP LHP140 CONT Vel= 50 % P_OLP30 Tool[1]:GUN C1 Base[1]:Actros ;%{PE}%R 4.1.16,%MKUKATPBASIS,%CMOVE,%VPTP,%P 1:PTP, 2:LHP140, 3:C_PTP, 5:50, 7:P_OLP30
$BWDSTART = FALSE
PDAT_ACT=PP_OLP30
BAS(#PTP_DAT)
FDAT_ACT=FLHP140
BAS(#FRAMES)
BAS(#VEL_PTP,50)
PTP XLHP140 C_PTP
;ENDFOLD

;FOLD ; SWP_60_4371;%{PE}%R2.2,%MKUKATPBASIS,%CCOMMENT,%VNORMAL,%P 2: SWP_60_4371
;ENDFOLD
;FOLD PTP p60_4371 PDAT18 SPOT Gun= 1 RETR CLS PgNo1= 117 ACTIVE= 1 Tool[1]:GUN C1 Base[1]:Actros ;%{PE}%R 4.1.12,%MKUKATPSPOT,%CSPOT,%VPTP,%P 1:PTP, 2:p60_4371, 3:, 5:100, 7:PDAT18, 10:1, 12:#FIRST, 14:#CLO, 16:117, 18:1, 20:0, 22:0, 24:1, 25:NORMAL
$BWDSTART = TRUE
PDAT_ACT=PPDAT18
BAS(#PTP_DAT)
FDAT_ACT=Fp60_4371
BAS(#FRAMES)
BAS(#VEL_PTP,PPDAT18.VEL)
S_ACT.GUN=1
S_ACT.PAIR=SDEFAULT.PAIR
S_ACT.RETR=#CLO
S_ACT.CLO_TM=1
S_ACT.PGNO1=117
S_ACT.PGNO2=SDEFAULT.PGNO2
S_ACT.PRESS1=SDEFAULT.PRESS1
S_ACT.PRESS2=SDEFAULT.PRESS2
S_READY=FALSE
PTP Xp60_4371
USERSPOT(#SPOT, S_ACT)
WAIT FOR S_READY
;ENDFOLD

;FOLD ; SWP_60_4369;%{PE}%R2.2,%MKUKATPBASIS,%CCOMMENT,%VNORMAL,%P 2: SWP_60_4369
;ENDFOLD
;FOLD PTP swp_60_4369 PDAT19 SPOT Gun= 1 RETR CLS PgNo1= 118 ACTIVE= 1 Tool[1]:GUN C1 Base[1]:Actros ;%{PE}%R 4.1.12,%MKUKATPSPOT,%CSPOT,%VPTP,%P 1:PTP, 2:swp_60_4369, 3:, 5:100, 7:PDAT19, 10:1, 12:#FIRST, 14:#CLO, 16:118, 18:1, 20:0, 22:0, 24:1, 25:NORMAL
$BWDSTART = TRUE
PDAT_ACT=PPDAT19
BAS(#PTP_DAT)
FDAT_ACT=Fswp_60_4369
BAS(#FRAMES)
BAS(#VEL_PTP,PPDAT19.VEL)
S_ACT.GUN=1
S_ACT.PAIR=SDEFAULT.PAIR
S_ACT.RETR=#CLO
S_ACT.CLO_TM=1
S_ACT.PGNO1=118
S_ACT.PGNO2=SDEFAULT.PGNO2
S_ACT.PRESS1=SDEFAULT.PRESS1
S_ACT.PRESS2=SDEFAULT.PRESS2
S_READY=FALSE
PTP Xswp_60_4369
USERSPOT(#SPOT, S_ACT)
WAIT FOR S_READY
;ENDFOLD

;FOLD ; SWP_60_4365;%{PE}%R2.2,%MKUKATPBASIS,%CCOMMENT,%VNORMAL,%P 2: SWP_60_4365
;ENDFOLD
;FOLD PTP swp_60_4365 PDAT20 SPOT Gun= 1 RETR CLS PgNo1= 119 ACTIVE= 1 Tool[1]:GUN C1 Base[1]:Actros ;%{PE}%R 4.1.12,%MKUKATPSPOT,%CSPOT,%VPTP,%P 1:PTP, 2:swp_60_4365, 3:, 5:100, 7:PDAT20, 10:1, 12:#FIRST, 14:#CLO, 16:119, 18:1, 20:0, 22:0, 24:1, 25:NORMAL
$BWDSTART = TRUE
PDAT_ACT=PPDAT20
BAS(#PTP_DAT)
FDAT_ACT=Fswp_60_4365
BAS(#FRAMES)
BAS(#VEL_PTP,PPDAT20.VEL)
S_ACT.GUN=1
S_ACT.PAIR=SDEFAULT.PAIR
S_ACT.RETR=#CLO
S_ACT.CLO_TM=1
S_ACT.PGNO1=119
S_ACT.PGNO2=SDEFAULT.PGNO2
S_ACT.PRESS1=SDEFAULT.PRESS1
S_ACT.PRESS2=SDEFAULT.PRESS2
S_READY=FALSE
PTP Xswp_60_4365
USERSPOT(#SPOT, S_ACT)
WAIT FOR S_READY
;ENDFOLD

;FOLD ; SWP_60_4361;%{PE}%R2.2,%MKUKATPBASIS,%CCOMMENT,%VNORMAL,%P 2: SWP_60_4361
;ENDFOLD
;FOLD PTP swp_60_4361 PDAT22 SPOT Gun= 1 RETR OPN PgNo1= 120 ACTIVE= 1 Tool[1]:GUN C1 Base[1]:Actros ;%{PE}%R 4.1.12,%MKUKATPSPOT,%CSPOT,%VPTP,%P 1:PTP, 2:swp_60_4361, 3:, 5:100, 7:PDAT22, 10:1, 12:#FIRST, 14:#OPN, 16:120, 18:1, 20:0, 22:0, 24:1, 25:NORMAL
$BWDSTART = TRUE
PDAT_ACT=PPDAT22
BAS(#PTP_DAT)
FDAT_ACT=Fswp_60_4361
BAS(#FRAMES)
BAS(#VEL_PTP,PPDAT22.VEL)
S_ACT.GUN=1
S_ACT.PAIR=SDEFAULT.PAIR
S_ACT.RETR=#OPN
S_ACT.CLO_TM=1
S_ACT.PGNO1=120
S_ACT.PGNO2=SDEFAULT.PGNO2
S_ACT.PRESS1=SDEFAULT.PRESS1
S_ACT.PRESS2=SDEFAULT.PRESS2
S_READY=FALSE
PTP Xswp_60_4361
USERSPOT(#SPOT, S_ACT)
WAIT FOR S_READY
;ENDFOLD

;FOLD PTP LHP145  Vel= 55 % P_OLP35 Tool[1]:GUN C1 Base[1]:Actros ;%{PE}%R 4.1.16,%MKUKATPBASIS,%CMOVE,%VPTP,%P 1:PTP, 2:LHP145, 3:, 5:55, 7:P_OLP35
$BWDSTART = FALSE
PDAT_ACT=PP_OLP35
BAS(#PTP_DAT)
FDAT_ACT=FLHP145
BAS(#FRAMES)
BAS(#VEL_PTP,55)
PTP XLHP145
;ENDFOLD
;FOLD PTP LHP150 CONT Vel= 60 % P_OLP36 Tool[1]:GUN C1 Base[1]:Actros ;%{PE}%R 4.1.16,%MKUKATPBASIS,%CMOVE,%VPTP,%P 1:PTP, 2:LHP150, 3:C_PTP, 5:60, 7:P_OLP36
$BWDSTART = FALSE
PDAT_ACT=PP_OLP36
BAS(#PTP_DAT)
FDAT_ACT=FLHP150
BAS(#FRAMES)
BAS(#VEL_PTP,60)
PTP XLHP150 C_PTP
;ENDFOLD
;FOLD PTP LHP155 CONT Vel= 65 % P_OLP37 Tool[1]:GUN C1 Base[1]:Actros ;%{PE}%R 4.1.16,%MKUKATPBASIS,%CMOVE,%VPTP,%P 1:PTP, 2:LHP155, 3:C_PTP, 5:65, 7:P_OLP37
$BWDSTART = FALSE
PDAT_ACT=PP_OLP37
BAS(#PTP_DAT)
FDAT_ACT=FLHP155
BAS(#FRAMES)
BAS(#VEL_PTP,65)
PTP XLHP155 C_PTP
;ENDFOLD
;FOLD PTP LHP160 CONT Vel= 65 % PDAT28 Tool[1]:GUN C1 Base[1]:Actros ;%{PE}%R 4.1.16,%MKUKATPBASIS,%CMOVE,%VPTP,%P 1:PTP, 2:LHP160, 3:C_PTP, 5:65, 7:PDAT28
$BWDSTART = FALSE
PDAT_ACT=PPDAT28
BAS(#PTP_DAT)
FDAT_ACT=FLHP160
BAS(#FRAMES)
BAS(#VEL_PTP,65)
PTP XLHP160 C_PTP
;ENDFOLD
;FOLD PTP LHP165 CONT Vel= 65 % PDAT44 Tool[1]:GUN C1 Base[1]:Actros ;%{PE}%R 4.1.16,%MKUKATPBASIS,%CMOVE,%VPTP,%P 1:PTP, 2:LHP165, 3:C_PTP, 5:65, 7:PDAT44
$BWDSTART = FALSE
PDAT_ACT=PPDAT44
BAS(#PTP_DAT)
FDAT_ACT=FLHP165
BAS(#FRAMES)
BAS(#VEL_PTP,65)
PTP XLHP165 C_PTP
;ENDFOLD
;FOLD PTP LHP170 CONT Vel= 60 % PDAT86 Tool[1]:GUN C1 Base[0];%{PE}%R 4.1.16,%MKUKATPBASIS,%CMOVE,%VPTP,%P 1:PTP, 2:LHP170, 3:C_PTP, 5:60, 7:PDAT86
$BWDSTART = FALSE
PDAT_ACT=PPDAT86
BAS(#PTP_DAT)
FDAT_ACT=FLHP170
BAS(#FRAMES)
BAS(#VEL_PTP,60)
PTP XLHP170 C_PTP
;ENDFOLD
;FOLD PTP LHP175 CONT Vel= 55 % PDAT87 Tool[1]:GUN C1 Base[0];%{PE}%R 4.1.16,%MKUKATPBASIS,%CMOVE,%VPTP,%P 1:PTP, 2:LHP175, 3:C_PTP, 5:55, 7:PDAT87
$BWDSTART = FALSE
PDAT_ACT=PPDAT87
BAS(#PTP_DAT)
FDAT_ACT=FLHP175
BAS(#FRAMES)
BAS(#VEL_PTP,55)
PTP XLHP175 C_PTP
;ENDFOLD
;FOLD PTP LHP180  Vel= 50 % PDAT88 Tool[1]:GUN C1 Base[0];%{PE}%R 4.1.16,%MKUKATPBASIS,%CMOVE,%VPTP,%P 1:PTP, 2:LHP180, 3:, 5:50, 7:PDAT88
$BWDSTART = FALSE
PDAT_ACT=PPDAT88
BAS(#PTP_DAT)
FDAT_ACT=FLHP180
BAS(#FRAMES)
BAS(#VEL_PTP,50)
PTP XLHP180
;ENDFOLD

;FOLD ; SWP 60_4357;%{PE}%R 4.1.16,%MKUKATPBASIS,%CCOMMENT,%VNORMAL,%P 2:SWP 60_4357
;ENDFOLD
;FOLD PTP swp_60_4357 PDAT89 SPOT Gun= 1 RETR CLS PgNo1= 121 ACTIVE= 1 Tool[1]:GUN C1 Base[1]:Actros ;%{PE}%R 4.1.12,%MKUKATPSPOT,%CSPOT,%VPTP,%P 1:PTP, 2:swp_60_4357, 3:, 5:100, 7:PDAT89, 10:1, 12:#FIRST, 14:#CLO, 16:121, 18:1, 20:0, 22:0, 24:1, 25:NORMAL
$BWDSTART = TRUE
PDAT_ACT=PPDAT89
BAS(#PTP_DAT)
FDAT_ACT=Fswp_60_4357
BAS(#FRAMES)
BAS(#VEL_PTP,PPDAT89.VEL)
S_ACT.GUN=1
S_ACT.PAIR=SDEFAULT.PAIR
S_ACT.RETR=#CLO
S_ACT.CLO_TM=1
S_ACT.PGNO1=121
S_ACT.PGNO2=SDEFAULT.PGNO2
S_ACT.PRESS1=SDEFAULT.PRESS1
S_ACT.PRESS2=SDEFAULT.PRESS2
S_READY=FALSE
PTP Xswp_60_4357
USERSPOT(#SPOT, S_ACT)
WAIT FOR S_READY
;ENDFOLD


;FOLD ; SWP 60_4355;%{PE}%R 4.1.16,%MKUKATPBASIS,%CCOMMENT,%VNORMAL,%P 2:SWP 60_4355
;ENDFOLD
;FOLD PTP swp_60_4355 PDAT90 SPOT Gun= 1 RETR CLS PgNo1= 122 ACTIVE= 1 Tool[1]:GUN C1 Base[1]:Actros ;%{PE}%R 4.1.12,%MKUKATPSPOT,%CSPOT,%VPTP,%P 1:PTP, 2:swp_60_4355, 3:, 5:100, 7:PDAT90, 10:1, 12:#FIRST, 14:#CLO, 16:122, 18:1, 20:0, 22:0, 24:1, 25:NORMAL
$BWDSTART = TRUE
PDAT_ACT=PPDAT90
BAS(#PTP_DAT)
FDAT_ACT=Fswp_60_4355
BAS(#FRAMES)
BAS(#VEL_PTP,PPDAT90.VEL)
S_ACT.GUN=1
S_ACT.PAIR=SDEFAULT.PAIR
S_ACT.RETR=#CLO
S_ACT.CLO_TM=1
S_ACT.PGNO1=122
S_ACT.PGNO2=SDEFAULT.PGNO2
S_ACT.PRESS1=SDEFAULT.PRESS1
S_ACT.PRESS2=SDEFAULT.PRESS2
S_READY=FALSE
PTP Xswp_60_4355
USERSPOT(#SPOT, S_ACT)
WAIT FOR S_READY
;ENDFOLD

;FOLD ; SWP_60_4351;%{PE}%R2.2,%MKUKATPBASIS,%CCOMMENT,%VNORMAL,%P 2: SWP_60_4351
;ENDFOLD
;FOLD PTP p60_4351 PDAT45 SPOT Gun= 1 RETR CLS PgNo1= 123 ACTIVE= 1 Tool[1]:GUN C1 Base[1]:Actros ;%{PE}%R 4.1.12,%MKUKATPSPOT,%CSPOT,%VPTP,%P 1:PTP, 2:p60_4351, 3:, 5:100, 7:PDAT45, 10:1, 12:#FIRST, 14:#CLO, 16:123, 18:1, 20:0, 22:0, 24:1, 25:NORMAL
$BWDSTART = TRUE
PDAT_ACT=PPDAT45
BAS(#PTP_DAT)
FDAT_ACT=Fp60_4351
BAS(#FRAMES)
BAS(#VEL_PTP,PPDAT45.VEL)
S_ACT.GUN=1
S_ACT.PAIR=SDEFAULT.PAIR
S_ACT.RETR=#CLO
S_ACT.CLO_TM=1
S_ACT.PGNO1=123
S_ACT.PGNO2=SDEFAULT.PGNO2
S_ACT.PRESS1=SDEFAULT.PRESS1
S_ACT.PRESS2=SDEFAULT.PRESS2
S_READY=FALSE
PTP Xp60_4351
USERSPOT(#SPOT, S_ACT)
WAIT FOR S_READY
;ENDFOLD

;FOLD ; SWP_60_4349;%{PE}%R2.2,%MKUKATPBASIS,%CCOMMENT,%VNORMAL,%P 2: SWP_60_4349
;ENDFOLD
;FOLD PTP p60_4349 PDAT46 SPOT Gun= 1 RETR OPN PgNo1= 124 ACTIVE= 1 Tool[1]:GUN C1 Base[1]:Actros ;%{PE}%R 4.1.12,%MKUKATPSPOT,%CSPOT,%VPTP,%P 1:PTP, 2:p60_4349, 3:, 5:100, 7:PDAT46, 10:1, 12:#FIRST, 14:#OPN, 16:124, 18:1, 20:0, 22:0, 24:1, 25:NORMAL
$BWDSTART = TRUE
PDAT_ACT=PPDAT46
BAS(#PTP_DAT)
FDAT_ACT=Fp60_4349
BAS(#FRAMES)
BAS(#VEL_PTP,PPDAT46.VEL)
S_ACT.GUN=1
S_ACT.PAIR=SDEFAULT.PAIR
S_ACT.RETR=#OPN
S_ACT.CLO_TM=1
S_ACT.PGNO1=124
S_ACT.PGNO2=SDEFAULT.PGNO2
S_ACT.PRESS1=SDEFAULT.PRESS1
S_ACT.PRESS2=SDEFAULT.PRESS2
S_READY=FALSE
PTP Xp60_4349
USERSPOT(#SPOT, S_ACT)
WAIT FOR S_READY
;ENDFOLD

;FOLD PTP LHP185 CONT Vel= 55 % PDAT47 Tool[1]:GUN C1 Base[1]:Actros ;%{PE}%R 4.1.16,%MKUKATPBASIS,%CMOVE,%VPTP,%P 1:PTP, 2:LHP185, 3:C_PTP, 5:55, 7:PDAT47
$BWDSTART = FALSE
PDAT_ACT=PPDAT47
BAS(#PTP_DAT)
FDAT_ACT=FLHP185
BAS(#FRAMES)
BAS(#VEL_PTP,55)
PTP XLHP185 C_PTP
;ENDFOLD

;FOLD ; swp_60_4345;%{PE}%R 4.1.16,%MKUKATPBASIS,%CCOMMENT,%VNORMAL,%P 2:swp_60_4345
;ENDFOLD
;FOLD PTP swp_60_4345 PDAT49 SPOT Gun= 1 RETR CLS PgNo1= 125 ACTIVE= 1 Tool[1]:GUN C1 Base[1]:Actros ;%{PE}%R 4.1.12,%MKUKATPSPOT,%CSPOT,%VPTP,%P 1:PTP, 2:swp_60_4345, 3:, 5:100, 7:PDAT49, 10:1, 12:#FIRST, 14:#CLO, 16:125, 18:1, 20:0, 22:0, 24:1, 25:NORMAL
$BWDSTART = TRUE
PDAT_ACT=PPDAT49
BAS(#PTP_DAT)
FDAT_ACT=Fswp_60_4345
BAS(#FRAMES)
BAS(#VEL_PTP,PPDAT49.VEL)
S_ACT.GUN=1
S_ACT.PAIR=SDEFAULT.PAIR
S_ACT.RETR=#CLO
S_ACT.CLO_TM=1
S_ACT.PGNO1=125
S_ACT.PGNO2=SDEFAULT.PGNO2
S_ACT.PRESS1=SDEFAULT.PRESS1
S_ACT.PRESS2=SDEFAULT.PRESS2
S_READY=FALSE
PTP Xswp_60_4345
USERSPOT(#SPOT, S_ACT)
WAIT FOR S_READY
;ENDFOLD

;FOLD ; SWP_60_4343;%{PE}%R2.2,%MKUKATPBASIS,%CCOMMENT,%VNORMAL,%P 2: SWP_60_4343
;ENDFOLD
;FOLD PTP p60_4343 PDAT50 SPOT Gun= 1 RETR CLS PgNo1= 126 ACTIVE= 1 Tool[1]:GUN C1 Base[1]:Actros ;%{PE}%R 4.1.12,%MKUKATPSPOT,%CSPOT,%VPTP,%P 1:PTP, 2:p60_4343, 3:, 5:100, 7:PDAT50, 10:1, 12:#FIRST, 14:#CLO, 16:126, 18:1, 20:0, 22:0, 24:1, 25:NORMAL
$BWDSTART = TRUE
PDAT_ACT=PPDAT50
BAS(#PTP_DAT)
FDAT_ACT=Fp60_4343
BAS(#FRAMES)
BAS(#VEL_PTP,PPDAT50.VEL)
S_ACT.GUN=1
S_ACT.PAIR=SDEFAULT.PAIR
S_ACT.RETR=#CLO
S_ACT.CLO_TM=1
S_ACT.PGNO1=126
S_ACT.PGNO2=SDEFAULT.PGNO2
S_ACT.PRESS1=SDEFAULT.PRESS1
S_ACT.PRESS2=SDEFAULT.PRESS2
S_READY=FALSE
PTP Xp60_4343
USERSPOT(#SPOT, S_ACT)
WAIT FOR S_READY
;ENDFOLD

;FOLD PTP LHP190 CONT Vel= 55 % P_OLP45 Tool[1]:GUN C1 Base[1]:Actros ;%{PE}%R 4.1.16,%MKUKATPBASIS,%CMOVE,%VPTP,%P 1:PTP, 2:LHP190, 3:C_PTP, 5:55, 7:P_OLP45
$BWDSTART = FALSE
PDAT_ACT=PP_OLP45
BAS(#PTP_DAT)
FDAT_ACT=FLHP190
BAS(#FRAMES)
BAS(#VEL_PTP,55)
PTP XLHP190 C_PTP
;ENDFOLD

;FOLD ; SWP_60_4339;%{PE}%R2.2,%MKUKATPBASIS,%CCOMMENT,%VNORMAL,%P 2: SWP_60_4339
;ENDFOLD
;FOLD PTP p60_4339 PDAT51 SPOT Gun= 1 RETR CLS PgNo1= 127 ACTIVE= 1 Tool[1]:GUN C1 Base[1]:Actros ;%{PE}%R 4.1.12,%MKUKATPSPOT,%CSPOT,%VPTP,%P 1:PTP, 2:p60_4339, 3:, 5:100, 7:PDAT51, 10:1, 12:#FIRST, 14:#CLO, 16:127, 18:1, 20:0, 22:0, 24:1, 25:NORMAL
$BWDSTART = TRUE
PDAT_ACT=PPDAT51
BAS(#PTP_DAT)
FDAT_ACT=Fp60_4339
BAS(#FRAMES)
BAS(#VEL_PTP,PPDAT51.VEL)
S_ACT.GUN=1
S_ACT.PAIR=SDEFAULT.PAIR
S_ACT.RETR=#CLO
S_ACT.CLO_TM=1
S_ACT.PGNO1=127
S_ACT.PGNO2=SDEFAULT.PGNO2
S_ACT.PRESS1=SDEFAULT.PRESS1
S_ACT.PRESS2=SDEFAULT.PRESS2
S_READY=FALSE
PTP Xp60_4339
USERSPOT(#SPOT, S_ACT)
WAIT FOR S_READY
;ENDFOLD

;FOLD ; SWP_60_4337;%{PE}%R2.2,%MKUKATPBASIS,%CCOMMENT,%VNORMAL,%P 2: SWP_60_4337
;ENDFOLD
;FOLD PTP p60_4337 PDAT52 SPOT Gun= 1 RETR CLS PgNo1= 128 ACTIVE= 1 Tool[1]:GUN C1 Base[1]:Actros ;%{PE}%R 4.1.12,%MKUKATPSPOT,%CSPOT,%VPTP,%P 1:PTP, 2:p60_4337, 3:, 5:100, 7:PDAT52, 10:1, 12:#FIRST, 14:#CLO, 16:128, 18:1, 20:0, 22:0, 24:1, 25:NORMAL
$BWDSTART = TRUE
PDAT_ACT=PPDAT52
BAS(#PTP_DAT)
FDAT_ACT=Fp60_4337
BAS(#FRAMES)
BAS(#VEL_PTP,PPDAT52.VEL)
S_ACT.GUN=1
S_ACT.PAIR=SDEFAULT.PAIR
S_ACT.RETR=#CLO
S_ACT.CLO_TM=1
S_ACT.PGNO1=128
S_ACT.PGNO2=SDEFAULT.PGNO2
S_ACT.PRESS1=SDEFAULT.PRESS1
S_ACT.PRESS2=SDEFAULT.PRESS2
S_READY=FALSE
PTP Xp60_4337
USERSPOT(#SPOT, S_ACT)
WAIT FOR S_READY
;ENDFOLD

;FOLD PTP LHP195 CONT Vel= 55 % PDAT81 Tool[1]:GUN C1 Base[1]:Actros ;%{PE}%R 4.1.16,%MKUKATPBASIS,%CMOVE,%VPTP,%P 1:PTP, 2:LHP195, 3:C_PTP, 5:55, 7:PDAT81
$BWDSTART = FALSE
PDAT_ACT=PPDAT81
BAS(#PTP_DAT)
FDAT_ACT=FLHP195
BAS(#FRAMES)
BAS(#VEL_PTP,55)
PTP XLHP195 C_PTP
;ENDFOLD
;FOLD PTP LHP200 CONT Vel= 55 % PDAT53 Tool[1]:GUN C1 Base[1]:Actros ;%{PE}%R 4.1.16,%MKUKATPBASIS,%CMOVE,%VPTP,%P 1:PTP, 2:LHP200, 3:C_PTP, 5:55, 7:PDAT53
$BWDSTART = FALSE
PDAT_ACT=PPDAT53
BAS(#PTP_DAT)
FDAT_ACT=FLHP200
BAS(#FRAMES)
BAS(#VEL_PTP,55)
PTP XLHP200 C_PTP
;ENDFOLD

;FOLD ; SWP_60_4333;%{PE}%R2.2,%MKUKATPBASIS,%CCOMMENT,%VNORMAL,%P 2: SWP_60_4333
;ENDFOLD
;FOLD PTP p60_4333 PDAT54 SPOT Gun= 1 RETR CLS PgNo1= 129 ACTIVE= 1 Tool[1]:GUN C1 Base[1]:Actros ;%{PE}%R 4.1.12,%MKUKATPSPOT,%CSPOT,%VPTP,%P 1:PTP, 2:p60_4333, 3:, 5:100, 7:PDAT54, 10:1, 12:#FIRST, 14:#CLO, 16:129, 18:1, 20:0, 22:0, 24:1, 25:NORMAL
$BWDSTART = TRUE
PDAT_ACT=PPDAT54
BAS(#PTP_DAT)
FDAT_ACT=Fp60_4333
BAS(#FRAMES)
BAS(#VEL_PTP,PPDAT54.VEL)
S_ACT.GUN=1
S_ACT.PAIR=SDEFAULT.PAIR
S_ACT.RETR=#CLO
S_ACT.CLO_TM=1
S_ACT.PGNO1=129
S_ACT.PGNO2=SDEFAULT.PGNO2
S_ACT.PRESS1=SDEFAULT.PRESS1
S_ACT.PRESS2=SDEFAULT.PRESS2
S_READY=FALSE
PTP Xp60_4333
USERSPOT(#SPOT, S_ACT)
WAIT FOR S_READY
;ENDFOLD

;FOLD ; SWP_60_4331;%{PE}%R2.2,%MKUKATPBASIS,%CCOMMENT,%VNORMAL,%P 2: SWP_60_4331
;ENDFOLD
;FOLD PTP p60_4331 PDAT55 SPOT Gun= 1 RETR CLS PgNo1= 130 ACTIVE= 1 Tool[1]:GUN C1 Base[1]:Actros ;%{PE}%R 4.1.12,%MKUKATPSPOT,%CSPOT,%VPTP,%P 1:PTP, 2:p60_4331, 3:, 5:100, 7:PDAT55, 10:1, 12:#FIRST, 14:#CLO, 16:130, 18:1, 20:0, 22:0, 24:1, 25:NORMAL
$BWDSTART = TRUE
PDAT_ACT=PPDAT55
BAS(#PTP_DAT)
FDAT_ACT=Fp60_4331
BAS(#FRAMES)
BAS(#VEL_PTP,PPDAT55.VEL)
S_ACT.GUN=1
S_ACT.PAIR=SDEFAULT.PAIR
S_ACT.RETR=#CLO
S_ACT.CLO_TM=1
S_ACT.PGNO1=130
S_ACT.PGNO2=SDEFAULT.PGNO2
S_ACT.PRESS1=SDEFAULT.PRESS1
S_ACT.PRESS2=SDEFAULT.PRESS2
S_READY=FALSE
PTP Xp60_4331
USERSPOT(#SPOT, S_ACT)
WAIT FOR S_READY
;ENDFOLD

;FOLD PTP LHP205 CONT Vel= 55 % PDAT82 Tool[1]:GUN C1 Base[1]:Actros ;%{PE}%R 4.1.16,%MKUKATPBASIS,%CMOVE,%VPTP,%P 1:PTP, 2:LHP205, 3:C_PTP, 5:55, 7:PDAT82
$BWDSTART = FALSE
PDAT_ACT=PPDAT82
BAS(#PTP_DAT)
FDAT_ACT=FLHP205
BAS(#FRAMES)
BAS(#VEL_PTP,55)
PTP XLHP205 C_PTP
;ENDFOLD

;FOLD ; SWP_60_4327;%{PE}%R2.2,%MKUKATPBASIS,%CCOMMENT,%VNORMAL,%P 2: SWP_60_4327
;ENDFOLD
;FOLD PTP p60_4327 PDAT56 SPOT Gun= 1 RETR CLS PgNo1= 131 ACTIVE= 1 Tool[1]:GUN C1 Base[1]:Actros ;%{PE}%R 4.1.12,%MKUKATPSPOT,%CSPOT,%VPTP,%P 1:PTP, 2:p60_4327, 3:, 5:100, 7:PDAT56, 10:1, 12:#FIRST, 14:#CLO, 16:131, 18:1, 20:0, 22:0, 24:1, 25:NORMAL
$BWDSTART = TRUE
PDAT_ACT=PPDAT56
BAS(#PTP_DAT)
FDAT_ACT=Fp60_4327
BAS(#FRAMES)
BAS(#VEL_PTP,PPDAT56.VEL)
S_ACT.GUN=1
S_ACT.PAIR=SDEFAULT.PAIR
S_ACT.RETR=#CLO
S_ACT.CLO_TM=1
S_ACT.PGNO1=131
S_ACT.PGNO2=SDEFAULT.PGNO2
S_ACT.PRESS1=SDEFAULT.PRESS1
S_ACT.PRESS2=SDEFAULT.PRESS2
S_READY=FALSE
PTP Xp60_4327
USERSPOT(#SPOT, S_ACT)
WAIT FOR S_READY
;ENDFOLD

;FOLD ; SWP_60_4325;%{PE}%R2.2,%MKUKATPBASIS,%CCOMMENT,%VNORMAL,%P 2: SWP_60_4325
;ENDFOLD
;FOLD PTP p60_4325 PDAT57 SPOT Gun= 1 RETR CLS PgNo1= 132 ACTIVE= 1 Tool[1]:GUN C1 Base[1]:Actros ;%{PE}%R 4.1.12,%MKUKATPSPOT,%CSPOT,%VPTP,%P 1:PTP, 2:p60_4325, 3:, 5:100, 7:PDAT57, 10:1, 12:#FIRST, 14:#CLO, 16:132, 18:1, 20:0, 22:0, 24:1, 25:NORMAL
$BWDSTART = TRUE
PDAT_ACT=PPDAT57
BAS(#PTP_DAT)
FDAT_ACT=Fp60_4325
BAS(#FRAMES)
BAS(#VEL_PTP,PPDAT57.VEL)
S_ACT.GUN=1
S_ACT.PAIR=SDEFAULT.PAIR
S_ACT.RETR=#CLO
S_ACT.CLO_TM=1
S_ACT.PGNO1=132
S_ACT.PGNO2=SDEFAULT.PGNO2
S_ACT.PRESS1=SDEFAULT.PRESS1
S_ACT.PRESS2=SDEFAULT.PRESS2
S_READY=FALSE
PTP Xp60_4325
USERSPOT(#SPOT, S_ACT)
WAIT FOR S_READY
;ENDFOLD

;FOLD PTP LHP210 CONT Vel= 55 % PDAT83 Tool[1]:GUN C1 Base[1]:Actros ;%{PE}%R 4.1.16,%MKUKATPBASIS,%CMOVE,%VPTP,%P 1:PTP, 2:LHP210, 3:C_PTP, 5:55, 7:PDAT83
$BWDSTART = FALSE
PDAT_ACT=PPDAT83
BAS(#PTP_DAT)
FDAT_ACT=FLHP210
BAS(#FRAMES)
BAS(#VEL_PTP,55)
PTP XLHP210 C_PTP
;ENDFOLD

;FOLD ; SWP_60_4321;%{PE}%R2.2,%MKUKATPBASIS,%CCOMMENT,%VNORMAL,%P 2: SWP_60_4321
;ENDFOLD
;FOLD PTP p60_4321 PDAT58 SPOT Gun= 1 RETR CLS PgNo1= 133 ACTIVE= 1 Tool[1]:GUN C1 Base[1]:Actros ;%{PE}%R 4.1.12,%MKUKATPSPOT,%CSPOT,%VPTP,%P 1:PTP, 2:p60_4321, 3:, 5:100, 7:PDAT58, 10:1, 12:#FIRST, 14:#CLO, 16:133, 18:1, 20:0, 22:0, 24:1, 25:NORMAL
$BWDSTART = TRUE
PDAT_ACT=PPDAT58
BAS(#PTP_DAT)
FDAT_ACT=Fp60_4321
BAS(#FRAMES)
BAS(#VEL_PTP,PPDAT58.VEL)
S_ACT.GUN=1
S_ACT.PAIR=SDEFAULT.PAIR
S_ACT.RETR=#CLO
S_ACT.CLO_TM=1
S_ACT.PGNO1=133
S_ACT.PGNO2=SDEFAULT.PGNO2
S_ACT.PRESS1=SDEFAULT.PRESS1
S_ACT.PRESS2=SDEFAULT.PRESS2
S_READY=FALSE
PTP Xp60_4321
USERSPOT(#SPOT, S_ACT)
WAIT FOR S_READY
;ENDFOLD

;FOLD ; SWP_60_4319;%{PE}%R2.2,%MKUKATPBASIS,%CCOMMENT,%VNORMAL,%P 2: SWP_60_4319
;ENDFOLD
;FOLD PTP p60_4319 PDAT59 SPOT Gun= 1 RETR CLS PgNo1= 134 ACTIVE= 1 Tool[1]:GUN C1 Base[1]:Actros ;%{PE}%R 4.1.12,%MKUKATPSPOT,%CSPOT,%VPTP,%P 1:PTP, 2:p60_4319, 3:, 5:100, 7:PDAT59, 10:1, 12:#FIRST, 14:#CLO, 16:134, 18:1, 20:0, 22:0, 24:1, 25:NORMAL
$BWDSTART = TRUE
PDAT_ACT=PPDAT59
BAS(#PTP_DAT)
FDAT_ACT=Fp60_4319
BAS(#FRAMES)
BAS(#VEL_PTP,PPDAT59.VEL)
S_ACT.GUN=1
S_ACT.PAIR=SDEFAULT.PAIR
S_ACT.RETR=#CLO
S_ACT.CLO_TM=1
S_ACT.PGNO1=134
S_ACT.PGNO2=SDEFAULT.PGNO2
S_ACT.PRESS1=SDEFAULT.PRESS1
S_ACT.PRESS2=SDEFAULT.PRESS2
S_READY=FALSE
PTP Xp60_4319
USERSPOT(#SPOT, S_ACT)
WAIT FOR S_READY
;ENDFOLD

;FOLD ; SWP_60_4315;%{PE}%R2.2,%MKUKATPBASIS,%CCOMMENT,%VNORMAL,%P 2: SWP_60_4315
;ENDFOLD
;FOLD PTP p60_4315 PDAT84 SPOT Gun= 1 RETR CLS PgNo1= 135 ACTIVE= 1 Tool[1]:GUN C1 Base[1]:Actros ;%{PE}%R 4.1.12,%MKUKATPSPOT,%CSPOT,%VPTP,%P 1:PTP, 2:p60_4315, 3:, 5:100, 7:PDAT84, 10:1, 12:#FIRST, 14:#CLO, 16:135, 18:1, 20:0, 22:0, 24:1, 25:NORMAL
$BWDSTART = TRUE
PDAT_ACT=PPDAT84
BAS(#PTP_DAT)
FDAT_ACT=Fp60_4315
BAS(#FRAMES)
BAS(#VEL_PTP,PPDAT84.VEL)
S_ACT.GUN=1
S_ACT.PAIR=SDEFAULT.PAIR
S_ACT.RETR=#CLO
S_ACT.CLO_TM=1
S_ACT.PGNO1=135
S_ACT.PGNO2=SDEFAULT.PGNO2
S_ACT.PRESS1=SDEFAULT.PRESS1
S_ACT.PRESS2=SDEFAULT.PRESS2
S_READY=FALSE
PTP Xp60_4315
USERSPOT(#SPOT, S_ACT)
WAIT FOR S_READY
;ENDFOLD

;FOLD ; SWP_60_4313;%{PE}%R2.2,%MKUKATPBASIS,%CCOMMENT,%VNORMAL,%P 2: SWP_60_4313
;ENDFOLD
;FOLD PTP p60_4313 PDAT61 SPOT Gun= 1 RETR CLS PgNo1= 136 ACTIVE= 1 Tool[1]:GUN C1 Base[1]:Actros ;%{PE}%R 4.1.12,%MKUKATPSPOT,%CSPOT,%VPTP,%P 1:PTP, 2:p60_4313, 3:, 5:100, 7:PDAT61, 10:1, 12:#FIRST, 14:#CLO, 16:136, 18:1, 20:0, 22:0, 24:1, 25:NORMAL
$BWDSTART = TRUE
PDAT_ACT=PPDAT61
BAS(#PTP_DAT)
FDAT_ACT=Fp60_4313
BAS(#FRAMES)
BAS(#VEL_PTP,PPDAT61.VEL)
S_ACT.GUN=1
S_ACT.PAIR=SDEFAULT.PAIR
S_ACT.RETR=#CLO
S_ACT.CLO_TM=1
S_ACT.PGNO1=136
S_ACT.PGNO2=SDEFAULT.PGNO2
S_ACT.PRESS1=SDEFAULT.PRESS1
S_ACT.PRESS2=SDEFAULT.PRESS2
S_READY=FALSE
PTP Xp60_4313
USERSPOT(#SPOT, S_ACT)
WAIT FOR S_READY
;ENDFOLD

;FOLD PTP LHP215 CONT Vel= 55 % PDAT85 Tool[1]:GUN C1 Base[1]:Actros ;%{PE}%R 4.1.16,%MKUKATPBASIS,%CMOVE,%VPTP,%P 1:PTP, 2:LHP215, 3:C_PTP, 5:55, 7:PDAT85
$BWDSTART = FALSE
PDAT_ACT=PPDAT85
BAS(#PTP_DAT)
FDAT_ACT=FLHP215
BAS(#FRAMES)
BAS(#VEL_PTP,55)
PTP XLHP215 C_PTP
;ENDFOLD

;FOLD ; SWP_60_4309;%{PE}%R2.2,%MKUKATPBASIS,%CCOMMENT,%VNORMAL,%P 2: SWP_60_4309
;ENDFOLD
;FOLD PTP p60_4309 PDAT62 SPOT Gun= 1 RETR CLS PgNo1= 137 ACTIVE= 1 Tool[1]:GUN C1 Base[1]:Actros ;%{PE}%R 4.1.12,%MKUKATPSPOT,%CSPOT,%VPTP,%P 1:PTP, 2:p60_4309, 3:, 5:100, 7:PDAT62, 10:1, 12:#FIRST, 14:#CLO, 16:137, 18:1, 20:0, 22:0, 24:1, 25:NORMAL
$BWDSTART = TRUE
PDAT_ACT=PPDAT62
BAS(#PTP_DAT)
FDAT_ACT=Fp60_4309
BAS(#FRAMES)
BAS(#VEL_PTP,PPDAT62.VEL)
S_ACT.GUN=1
S_ACT.PAIR=SDEFAULT.PAIR
S_ACT.RETR=#CLO
S_ACT.CLO_TM=1
S_ACT.PGNO1=137
S_ACT.PGNO2=SDEFAULT.PGNO2
S_ACT.PRESS1=SDEFAULT.PRESS1
S_ACT.PRESS2=SDEFAULT.PRESS2
S_READY=FALSE
PTP Xp60_4309
USERSPOT(#SPOT, S_ACT)
WAIT FOR S_READY
;ENDFOLD

;FOLD ; SWP_60_4307;%{PE}%R 4.1.16,%MKUKATPBASIS,%CCOMMENT,%VNORMAL,%P 2:SWP_60_4307
;ENDFOLD
;FOLD PTP p60_4307 PDAT92 SPOT Gun= 1 RETR CLS PgNo1= 137 ACTIVE= 1 Tool[1]:GUN C1 Base[1]:Actros ;%{PE}%R 4.1.12,%MKUKATPSPOT,%CSPOT,%VPTP,%P 1:PTP, 2:p60_4307, 3:, 5:70, 7:PDAT92, 10:1, 12:#FIRST, 14:#CLO, 16:137, 18:1, 20:0, 22:0, 24:1, 25:NORMAL
$BWDSTART = TRUE
PDAT_ACT=PPDAT92
BAS(#PTP_DAT)
FDAT_ACT=Fp60_4307
BAS(#FRAMES)
BAS(#VEL_PTP,PPDAT92.VEL)
S_ACT.GUN=1
S_ACT.PAIR=SDEFAULT.PAIR
S_ACT.RETR=#CLO
S_ACT.CLO_TM=1
S_ACT.PGNO1=137
S_ACT.PGNO2=SDEFAULT.PGNO2
S_ACT.PRESS1=SDEFAULT.PRESS1
S_ACT.PRESS2=SDEFAULT.PRESS2
S_READY=FALSE
PTP Xp60_4307
USERSPOT(#SPOT, S_ACT)
WAIT FOR S_READY
;ENDFOLD

;FOLD ; SWP_60_4305;%{PE}%R2.2,%MKUKATPBASIS,%CCOMMENT,%VNORMAL,%P 2: SWP_60_4305
;ENDFOLD
;FOLD PTP p60_4305 PDAT64 SPOT Gun= 1 RETR CLS PgNo1= 138 ACTIVE= 1 Tool[1]:GUN C1 Base[1]:Actros ;%{PE}%R 4.1.12,%MKUKATPSPOT,%CSPOT,%VPTP,%P 1:PTP, 2:p60_4305, 3:, 5:100, 7:PDAT64, 10:1, 12:#FIRST, 14:#CLO, 16:138, 18:1, 20:0, 22:0, 24:1, 25:NORMAL
$BWDSTART = TRUE
PDAT_ACT=PPDAT64
BAS(#PTP_DAT)
FDAT_ACT=Fp60_4305
BAS(#FRAMES)
BAS(#VEL_PTP,PPDAT64.VEL)
S_ACT.GUN=1
S_ACT.PAIR=SDEFAULT.PAIR
S_ACT.RETR=#CLO
S_ACT.CLO_TM=1
S_ACT.PGNO1=138
S_ACT.PGNO2=SDEFAULT.PGNO2
S_ACT.PRESS1=SDEFAULT.PRESS1
S_ACT.PRESS2=SDEFAULT.PRESS2
S_READY=FALSE
PTP Xp60_4305
USERSPOT(#SPOT, S_ACT)
WAIT FOR S_READY
;ENDFOLD

;FOLD ; SWP_60_4303;%{PE}%R2.2,%MKUKATPBASIS,%CCOMMENT,%VNORMAL,%P 2: SWP_60_4303
;ENDFOLD
;FOLD PTP p60_4303 PDAT65 SPOT Gun= 1 RETR CLS PgNo1= 139 ACTIVE= 1 Tool[1]:GUN C1 Base[1]:Actros ;%{PE}%R 4.1.12,%MKUKATPSPOT,%CSPOT,%VPTP,%P 1:PTP, 2:p60_4303, 3:, 5:100, 7:PDAT65, 10:1, 12:#FIRST, 14:#CLO, 16:139, 18:1, 20:0, 22:0, 24:1, 25:NORMAL
$BWDSTART = TRUE
PDAT_ACT=PPDAT65
BAS(#PTP_DAT)
FDAT_ACT=Fp60_4303
BAS(#FRAMES)
BAS(#VEL_PTP,PPDAT65.VEL)
S_ACT.GUN=1
S_ACT.PAIR=SDEFAULT.PAIR
S_ACT.RETR=#CLO
S_ACT.CLO_TM=1
S_ACT.PGNO1=139
S_ACT.PGNO2=SDEFAULT.PGNO2
S_ACT.PRESS1=SDEFAULT.PRESS1
S_ACT.PRESS2=SDEFAULT.PRESS2
S_READY=FALSE
PTP Xp60_4303
USERSPOT(#SPOT, S_ACT)
WAIT FOR S_READY
;ENDFOLD

;FOLD ; SWP_60_4301;%{PE}%R2.2,%MKUKATPBASIS,%CCOMMENT,%VNORMAL,%P 2: SWP_60_4301
;ENDFOLD
;FOLD PTP p60_4301 PDAT66 SPOT Gun= 1 RETR CLS PgNo1= 139 ACTIVE= 1 Tool[1]:GUN C1 Base[1]:Actros ;%{PE}%R 4.1.12,%MKUKATPSPOT,%CSPOT,%VPTP,%P 1:PTP, 2:p60_4301, 3:, 5:100, 7:PDAT66, 10:1, 12:#FIRST, 14:#CLO, 16:139, 18:1, 20:0, 22:0, 24:1, 25:NORMAL
$BWDSTART = TRUE
PDAT_ACT=PPDAT66
BAS(#PTP_DAT)
FDAT_ACT=Fp60_4301
BAS(#FRAMES)
BAS(#VEL_PTP,PPDAT66.VEL)
S_ACT.GUN=1
S_ACT.PAIR=SDEFAULT.PAIR
S_ACT.RETR=#CLO
S_ACT.CLO_TM=1
S_ACT.PGNO1=139
S_ACT.PGNO2=SDEFAULT.PGNO2
S_ACT.PRESS1=SDEFAULT.PRESS1
S_ACT.PRESS2=SDEFAULT.PRESS2
S_READY=FALSE
PTP Xp60_4301
USERSPOT(#SPOT, S_ACT)
WAIT FOR S_READY
;ENDFOLD

;FOLD ; SWP_60_4300;%{PE}%R2.2,%MKUKATPBASIS,%CCOMMENT,%VNORMAL,%P 2: SWP_60_4300
;ENDFOLD
;FOLD PTP p60_4300 PDAT67 SPOT Gun= 1 RETR OPN PgNo1= 140 ACTIVE= 1 Tool[1]:GUN C1 Base[1]:Actros ;%{PE}%R 4.1.12,%MKUKATPSPOT,%CSPOT,%VPTP,%P 1:PTP, 2:p60_4300, 3:, 5:100, 7:PDAT67, 10:1, 12:#FIRST, 14:#OPN, 16:140, 18:1, 20:0, 22:0, 24:1, 25:NORMAL
$BWDSTART = TRUE
PDAT_ACT=PPDAT67
BAS(#PTP_DAT)
FDAT_ACT=Fp60_4300
BAS(#FRAMES)
BAS(#VEL_PTP,PPDAT67.VEL)
S_ACT.GUN=1
S_ACT.PAIR=SDEFAULT.PAIR
S_ACT.RETR=#OPN
S_ACT.CLO_TM=1
S_ACT.PGNO1=140
S_ACT.PGNO2=SDEFAULT.PGNO2
S_ACT.PRESS1=SDEFAULT.PRESS1
S_ACT.PRESS2=SDEFAULT.PRESS2
S_READY=FALSE
PTP Xp60_4300
USERSPOT(#SPOT, S_ACT)
WAIT FOR S_READY
;ENDFOLD

;FOLD PTP LHP220 CONT Vel= 55 % P_OLP62 Tool[1]:GUN C1 Base[1]:Actros ;%{PE}%R 4.1.16,%MKUKATPBASIS,%CMOVE,%VPTP,%P 1:PTP, 2:LHP220, 3:C_PTP, 5:55, 7:P_OLP62
$BWDSTART = FALSE
PDAT_ACT=PP_OLP62
BAS(#PTP_DAT)
FDAT_ACT=FLHP220
BAS(#FRAMES)
BAS(#VEL_PTP,55)
PTP XLHP220 C_PTP
;ENDFOLD
;FOLD PTP LHP225 CONT Vel= 65 % P_OLP63 Tool[1]:GUN C1 Base[1]:Actros ;%{PE}%R 4.1.16,%MKUKATPBASIS,%CMOVE,%VPTP,%P 1:PTP, 2:LHP225, 3:C_PTP, 5:65, 7:P_OLP63
$BWDSTART = FALSE
PDAT_ACT=PP_OLP63
BAS(#PTP_DAT)
FDAT_ACT=FLHP225
BAS(#FRAMES)
BAS(#VEL_PTP,65)
PTP XLHP225 C_PTP
;ENDFOLD
;FOLD PTP LHP230 CONT Vel= 65 % P_OLP64 Tool[1]:GUN C1 Base[1]:Actros ;%{PE}%R 4.1.16,%MKUKATPBASIS,%CMOVE,%VPTP,%P 1:PTP, 2:LHP230, 3:C_PTP, 5:65, 7:P_OLP64
$BWDSTART = FALSE
PDAT_ACT=PP_OLP64
BAS(#PTP_DAT)
FDAT_ACT=FLHP230
BAS(#FRAMES)
BAS(#VEL_PTP,65)
PTP XLHP230 C_PTP
;ENDFOLD
;FOLD PTP LHP235 CONT Vel= 70 % P_OLP65 Tool[1]:GUN C1 Base[1]:Actros ;%{PE}%R 4.1.16,%MKUKATPBASIS,%CMOVE,%VPTP,%P 1:PTP, 2:LHP235, 3:C_PTP, 5:70, 7:P_OLP65
$BWDSTART = FALSE
PDAT_ACT=PP_OLP65
BAS(#PTP_DAT)
FDAT_ACT=FLHP235
BAS(#FRAMES)
BAS(#VEL_PTP,70)
PTP XLHP235 C_PTP
;ENDFOLD

;FOLD ; END INTERLOCK WITH R2;%{PE}%R 4.1.16,%MKUKATPBASIS,%CCOMMENT,%VNORMAL,%P 2:END INTERLOCK WITH R2
;ENDFOLD
;FOLD Kollision.Ueberwachung_2_Aus ;%{PE}%MKUKATPUSER
COLLSTOP( 2, 2 )
;ENDFOLD

;FOLD PTP LHP240 CONT Vel= 70 % PDAT91 Tool[1]:GUN C1 Base[1]:Actros ;%{PE}%R 4.1.16,%MKUKATPBASIS,%CMOVE,%VPTP,%P 1:PTP, 2:LHP240, 3:C_PTP, 5:70, 7:PDAT91
$BWDSTART = FALSE
PDAT_ACT=PPDAT91
BAS(#PTP_DAT)
FDAT_ACT=FLHP240
BAS(#FRAMES)
BAS(#VEL_PTP,70)
PTP XLHP240 C_PTP
;ENDFOLD

;FOLD OUT 3331 'R1_Soldando' State=FALSE ;%{PE}%R 8.2.20,%MKUKATPBASIS,%COUT,%VOUTX,%P 2:3331, 3:R1_Soldando, 5:FALSE, 6:
$OUT[3331]=FALSE
;ENDFOLD
;FOLD OUT 3369 'Area de Solda' State=TRUE ;%{PE}%R 8.2.20,%MKUKATPBASIS,%COUT,%VOUTX,%P 2:3369, 3:Area de Solda, 5:TRUE, 6:
$OUT[3369]=TRUE
;ENDFOLD
;FOLD PULSE 3334 'R1_Solda Respot OK' State=TRUE CONT Time=3 sec;%{PE}%R 8.2.20,%MKUKATPBASIS,%COUT,%VPULSE,%P 2:3334, 3:R1_Solda Respot OK, 5:TRUE, 6:CONTINUE, 8:3
CONTINUE
PULSE($OUT[3334], TRUE,3)
;ENDFOLD

;FOLD PTP LHP245 CONT Vel= 70 % P_OLP66 Tool[1]:GUN C1 Base[1]:Actros ;%{PE}%R 4.1.16,%MKUKATPBASIS,%CMOVE,%VPTP,%P 1:PTP, 2:LHP245, 3:C_PTP, 5:70, 7:P_OLP66
$BWDSTART = FALSE
PDAT_ACT=PP_OLP66
BAS(#PTP_DAT)
FDAT_ACT=FLHP245
BAS(#FRAMES)
BAS(#VEL_PTP,70)
PTP XLHP245 C_PTP
;ENDFOLD
;FOLD PTP LHP250 CONT Vel= 70 % P_OLP67 Tool[1]:GUN C1 Base[1]:Actros ;%{PE}%R 4.1.16,%MKUKATPBASIS,%CMOVE,%VPTP,%P 1:PTP, 2:LHP250, 3:C_PTP, 5:70, 7:P_OLP67
$BWDSTART = FALSE
PDAT_ACT=PP_OLP67
BAS(#PTP_DAT)
FDAT_ACT=FLHP250
BAS(#FRAMES)
BAS(#VEL_PTP,70)
PTP XLHP250 C_PTP
;ENDFOLD

;FOLD PTP HOME  Vel= 80 % DEFAULT;%{PE}%R 4.1.16,%MKUKATPBASIS,%CMOVE,%VPTP,%P 1:PTP, 2:HOME, 3:, 5:80, 7:DEFAULT
$BWDSTART = FALSE
PDAT_ACT=PDEFAULT
BAS(#PTP_DAT)
FDAT_ACT=FHOME
BAS(#FRAMES)
BAS(#VEL_PTP,80)
$H_POS=XHOME
PTP XHOME
;ENDFOLD

IF (NOT(GHOST())) THEN
IF FraesAnf(1) THEN
  f_Fraes_1()
ENDIF
ENDIF

END

--- ps_601s1.dat ---
&ACCESS RVO2
&REL 23
&COMMENT Solda Respot C1 STB
DEFDAT  ps_601s1
;FOLD EXTERNAL DECLARATIONS;%{PE}%MKUKATPBASIS,%CEXT,%VCOMMON,%P
;FOLD GRIPPERTECH EXT
EXT  H50 (INT  :IN,INT  :IN,INT  :IN,GRP_TYP  :IN )
;ENDFOLD (GRIPPERTECH EXT)
;FOLD SPOTTECH EXT
EXT  USERSPOT (S_COMMAND  :IN,SPOT_TYPE  :IN )
;ENDFOLD (SPOTTECH EXT)
;FOLD BASISTECH EXT;%{PE}%MKUKATPBASIS,%CEXT,%VEXT,%P
EXT  BAS (BAS_COMMAND  :IN,REAL  :IN )
DECL INT SUCCESS
;ENDFOLD (BASISTECH EXT)
;FOLD USER EXT;%{E}%MKUKATPUSER,%CEXT,%VEXT,%P
;Make your modifications here

;ENDFOLD (USER EXT)
;ENDFOLD (EXTERNAL DECLARATIONS)

;# ============ START PATH : swp_p13060r1_stb_respot_c1 =============
DECL PDAT PP_OLP1={VEL 70.0,ACC 100.0,APO_DIST 0.0}
DECL FDAT FLHP010={TOOL_NO 1,BASE_NO 1,IPO_FRAME #BASE}
DECL PDAT PP_OLP2={VEL 100.0,ACC 100.0,APO_DIST 100.0}
DECL E6POS XLHP010={X 522.541016,Y -1798.11096,Z 280.665009,A 65.223999,B -21.2217999,C 44.3135986,S 2,T 35}
DECL FDAT FLHP015={TOOL_NO 1,BASE_NO 1,IPO_FRAME #BASE}
DECL PDAT PP_OLP3={VEL 100.0,ACC 100.0,APO_DIST 100.0}
DECL E6POS XLHP015={X 1400.79004,Y -1392.66394,Z 189.25,A 160.815994,B -71.8742981,C -72.1356964,S 2,T 35}
DECL FDAT FLHP020={TOOL_NO 1,BASE_NO 1,IPO_FRAME #BASE}
DECL PDAT PP_OLP4={VEL 100.0,ACC 100.0,APO_DIST 100.0}
DECL E6POS XLHP020={X 1485.43701,Y -1354.09595,Z -82.8130035,A 160.820297,B -71.873703,C -72.1393967,S 2,T 35}
DECL FDAT FLHP035={TOOL_NO 1,BASE_NO 1,IPO_FRAME #BASE}
DECL PDAT PP_OLP10={VEL 100.0,ACC 100.0,APO_DIST 100.0}
DECL E6POS XLHP035={X 1552.40601,Y -1264.67395,Z -66.6750031,A 18.0507908,B -82.7117233,C 75.4039383,S 2,T 35,E1 0.0,E2 0.0,E3 0.0,E4 0.0,E5 0.0,E6 0.0}
DECL FDAT FLHP070={TOOL_NO 1,BASE_NO 1,IPO_FRAME #BASE}
DECL PDAT PP_OLP12={VEL 100.0,ACC 100.0,APO_DIST 100.0}
DECL E6POS XLHP070={X 898.058777,Y -1607.94604,Z 736.711121,A -156.667297,B 31.9564304,C -84.0474472,S 2,T 3,E1 0.0,E2 0.0,E3 0.0,E4 0.0,E5 0.0,E6 0.0}
DECL FDAT FLHP075={TOOL_NO 1,BASE_NO 1,IPO_FRAME #BASE}
DECL PDAT PP_OLP13={VEL 100.0,ACC 100.0,APO_DIST 100.0}
DECL E6POS XLHP075={X 1169.72998,Y -1309.74695,Z 1575.08398,A 8.02140045,B 44.3081017,C 90.0,S 2,T 3}
DECL FDAT FLHP095={TOOL_NO 1,BASE_NO 1,IPO_FRAME #BASE}
DECL PDAT PP_OLP22={VEL 100.0,ACC 100.0,APO_DIST 0.0}
DECL E6POS XLHP095={X 1306.92004,Y -1063.49194,Z 1573.828,A 0.114962198,B 44.9941711,C 90.0060425,S 2,T 3,E1 0.0,E2 0.0,E3 0.0,E4 0.0,E5 0.0,E6 0.0}
DECL FDAT FLHP100={TOOL_NO 1,BASE_NO 1,IPO_FRAME #BASE}
DECL PDAT PP_OLP23={VEL 100.0,ACC 100.0,APO_DIST 100.0}
DECL E6POS XLHP100={X 1307.46594,Y -1346.25903,Z 1573.80701,A 0.114951402,B 44.9941711,C 90.0060272,S 2,T 3,E1 0.0,E2 0.0,E3 0.0,E4 0.0,E5 0.0,E6 0.0}
DECL FDAT FLHP105={TOOL_NO 1,BASE_NO 1,IPO_FRAME #BASE}
DECL PDAT PP_OLP24={VEL 100.0,ACC 100.0,APO_DIST 0.0}
DECL E6POS XLHP105={X 962.844971,Y -1334.99597,Z 1566.15601,A 180.0,B 46.2584991,C -90.0,S 2,T 3}
DECL FDAT FLHP110={TOOL_NO 1,BASE_NO 1,IPO_FRAME #BASE}
DECL PDAT PP_OLP25={VEL 100.0,ACC 100.0,APO_DIST 100.0}
DECL E6POS XLHP110={X 1778.90796,Y -2207.25195,Z 26.1790009,A -6.18400002,B 23.5095997,C 33.8945999,S 2,T 3}
DECL FDAT FLHP115={TOOL_NO 1,BASE_NO 1,IPO_FRAME #BASE}
DECL PDAT PP_OLP26={VEL 100.0,ACC 100.0,APO_DIST 100.0}
DECL E6POS XLHP115={X 2934.2229,Y -1484.28101,Z 26.1779995,A -66.0009003,B 23.5097008,C 33.8945999,S 2,T 3}
DECL FDAT FLHP125={TOOL_NO 1,BASE_NO 1,IPO_FRAME #BASE}
DECL PDAT PP_OLP27={VEL 100.0,ACC 100.0,APO_DIST 100.0}
DECL E6POS XLHP125={X 2545.36499,Y -771.27002,Z -167.815994,A -157.145294,B -17.1744995,C -18.4382,S 2,T 10}
DECL FDAT FLHP130={TOOL_NO 1,BASE_NO 1,IPO_FRAME #BASE}
DECL PDAT PP_OLP28={VEL 100.0,ACC 100.0,APO_DIST 100.0}
DECL E6POS XLHP130={X 1803.36096,Y -1070.38,Z 128.423996,A 169.254898,B -58.8148003,C 15.0047998,S 2,T 10}
DECL FDAT FLHP135={TOOL_NO 1,BASE_NO 1,IPO_FRAME #BASE}
DECL PDAT PP_OLP29={VEL 100.0,ACC 100.0,APO_DIST 100.0}
DECL E6POS XLHP135={X 1754.26904,Y -1045.44495,Z -70.9319992,A 94.819603,B -27.4731998,C 81.3091965,S 2,T 10}
DECL FDAT FLHP140={TOOL_NO 1,BASE_NO 1,IPO_FRAME #BASE}
DECL PDAT PP_OLP30={VEL 100.0,ACC 100.0,APO_DIST 100.0}
DECL E6POS XLHP140={X 1565.26904,Y -1045.44202,Z -70.9440002,A 94.8190002,B -27.4722004,C 81.3095016,S 2,T 10}
DECL FDAT FLHP145={TOOL_NO 1,BASE_NO 1,IPO_FRAME #BASE}
DECL PDAT PP_OLP35={VEL 100.0,ACC 100.0,APO_DIST 100.0}
DECL E6POS XLHP145={X 1559.547,Y -855.092407,Z -68.3633194,A 90.0005722,B 0.879426718,C 89.9992065,S 2,T 10,E1 0.0,E2 0.0,E3 0.0,E4 0.0,E5 0.0,E6 0.0}
DECL FDAT FLHP150={TOOL_NO 1,BASE_NO 1,IPO_FRAME #BASE}
DECL PDAT PP_OLP36={VEL 100.0,ACC 100.0,APO_DIST 100.0}
DECL E6POS XLHP150={X 1780.19397,Y -855.191223,Z -73.0292969,A 90.0003662,B 1.68043494,C 89.9991531,S 2,T 10,E1 0.0,E2 0.0,E3 0.0,E4 0.0,E5 0.0,E6 0.0}
DECL FDAT FLHP155={TOOL_NO 1,BASE_NO 1,IPO_FRAME #BASE}
DECL PDAT PP_OLP37={VEL 100.0,ACC 100.0,APO_DIST 100.0}
DECL E6POS XLHP155={X 1803.36096,Y -1070.38,Z 128.423996,A 169.254898,B -58.8148003,C 15.0047998,S 2,T 10}
DECL FDAT FLHP190={TOOL_NO 1,BASE_NO 1,IPO_FRAME #BASE}
DECL PDAT PP_OLP45={VEL 100.0,ACC 100.0,APO_DIST 0.0}
DECL E6POS XLHP190={X 1559.67505,Y -562.556274,Z 97.9280319,A -92.2449036,B -8.1948061,C -91.3425827,S 2,T 10,E1 0.0,E2 0.0,E3 0.0,E4 0.0,E5 0.0,E6 0.0}
DECL FDAT FLHP220={TOOL_NO 1,BASE_NO 1,IPO_FRAME #BASE}
DECL PDAT PP_OLP62={VEL 100.0,ACC 100.0,APO_DIST 100.0}
DECL E6POS XLHP220={X 1562.922,Y -0.708318412,Z 303.973511,A 83.1230927,B -60.6636505,C 94.3970871,S 2,T 10,E1 0.0,E2 0.0,E3 0.0,E4 0.0,E5 0.0,E6 0.0}
DECL FDAT FLHP225={TOOL_NO 1,BASE_NO 1,IPO_FRAME #BASE}
DECL PDAT PP_OLP63={VEL 100.0,ACC 100.0,APO_DIST 100.0}
DECL E6POS XLHP225={X 1752.61804,Y -51.1363182,Z 217.937393,A 162.001602,B -76.6891785,C 10.8350096,S 2,T 10,E1 0.0,E2 0.0,E3 0.0,E4 0.0,E5 0.0,E6 0.0}
DECL FDAT FLHP230={TOOL_NO 1,BASE_NO 1,IPO_FRAME #BASE}
DECL PDAT PP_OLP64={VEL 100.0,ACC 100.0,APO_DIST 100.0}
DECL E6POS XLHP230={X 2472.78491,Y -503.103088,Z -40.6362801,A -158.060196,B -14.5187302,C -31.7777004,S 2,T 10,E1 0.0,E2 0.0,E3 0.0,E4 0.0,E5 0.0,E6 0.0}
DECL FDAT FLHP235={TOOL_NO 1,BASE_NO 1,IPO_FRAME #BASE}
DECL PDAT PP_OLP65={VEL 100.0,ACC 100.0,APO_DIST 100.0}
DECL E6POS XLHP235={X 2899.50903,Y -1348.60901,Z -259.222198,A -159.819107,B -6.23635387,C -5.25122118,S 2,T 10,E1 0.0,E2 0.0,E3 0.0,E4 0.0,E5 0.0,E6 0.0}
DECL FDAT FLHP245={TOOL_NO 1,BASE_NO 1,IPO_FRAME #BASE}
DECL PDAT PP_OLP66={VEL 100.0,ACC 100.0,APO_DIST 100.0}
DECL E6POS XLHP245={X 1820.70203,Y -2027.24597,Z -233.501694,A -159.819107,B -6.23635387,C -5.25117207,S 2,T 11,E1 0.0,E2 0.0,E3 0.0,E4 0.0,E5 0.0,E6 0.0}
DECL FDAT FLHP250={TOOL_NO 1,BASE_NO 1,IPO_FRAME #BASE}
DECL PDAT PP_OLP67={VEL 100.0,ACC 100.0,APO_DIST 0.0}
DECL E6POS XLHP250={X 1283.02197,Y -2788.74805,Z -174.021103,A -134.645203,B -8.80581188,C -10.8908596,S 2,T 11,E1 0.0,E2 0.0,E3 0.0,E4 0.0,E5 0.0,E6 0.0}
DECL SPOT_SUGG_T LAST_SPOT={GUN[] "1                       ",RETR_CMD[] "#CLO                    ",CHOISE[] "#FIRST                  ",CLO_TM[] "1                       ",PGNO1[] "137                     ",PRESS1[] "0                       ",PGNO2[] "1                       ",PRESS2[] "0                       ",SPOT_PARAMS[] "NORMAL                  "}
DECL E6POS XLHP025={X 1475.17896,Y -1119.72302,Z -85.4240265,A 160.822205,B -71.8717575,C -67.4135132,S 2,T 35,E1 0.0,E2 0.0,E3 0.0,E4 0.0,E5 0.0,E6 0.0}
DECL FDAT FLHP025={TOOL_NO 1,BASE_NO 1,IPO_FRAME #BASE}
DECL PDAT PPDAT1={VEL 50.0,ACC 100.0,APO_DIST 100.0}
DECL PDAT PPDAT3={VEL 50.0,ACC 100.0,APO_DIST 100.0}
DECL PDAT PPDAT4={VEL 50.0,ACC 100.0,APO_DIST 100.0}
DECL PDAT PPDAT5={VEL 50.0,ACC 100.0,APO_DIST 100.0}
DECL E6POS XLHP060={X 895.5448,Y -1367.26599,Z 692.181824,A -0.546224773,B -61.93647,C 95.6030121,S 2,T 35,E1 0.0,E2 0.0,E3 0.0,E4 0.0,E5 0.0,E6 0.0}
DECL FDAT FLHP060={TOOL_NO 1,BASE_NO 1,IPO_FRAME #BASE}
DECL PDAT PPDAT7={VEL 100.0,ACC 100.0,APO_DIST 100.0}
DECL E6POS XLHP065={X 374.468109,Y -1805.93506,Z -88.8473129,A 51.4655914,B -41.4590607,C 52.5988808,S 2,T 35,E1 0.0,E2 0.0,E3 0.0,E4 0.0,E5 0.0,E6 0.0}
DECL FDAT FLHP065={TOOL_NO 1,BASE_NO 1,IPO_FRAME #BASE}
DECL PDAT PPDAT8={VEL 100.0,ACC 100.0,APO_DIST 100.0}
DECL E6POS XLHP080={X 1300.78003,Y -1047.08704,Z 1577.14502,A 0.000244454714,B 44.3083382,C 90.0002365,S 2,T 3,E1 0.0,E2 0.0,E3 0.0,E4 0.0,E5 0.0,E6 0.0}
DECL FDAT FLHP080={TOOL_NO 1,BASE_NO 1,IPO_FRAME #BASE}
DECL PDAT PPDAT9={VEL 65.0,ACC 100.0,APO_DIST 100.0}
DECL E6POS XLHP085={X 1231.80396,Y -1059.99695,Z 1494.09497,A -0.0159092806,B 44.3085518,C 89.9878387,S 2,T 3,E1 0.0,E2 0.0,E3 0.0,E4 0.0,E5 0.0,E6 0.0}
DECL FDAT FLHP085={TOOL_NO 1,BASE_NO 1,IPO_FRAME #BASE}
DECL PDAT PPDAT10={VEL 60.0,ACC 100.0,APO_DIST 100.0}
DECL PDAT PPDAT11={VEL 55.0,ACC 100.0,APO_DIST 100.0}
DECL PDAT PPDAT12={VEL 55.0,ACC 100.0,APO_DIST 100.0}
DECL PDAT PPDAT13={VEL 55.0,ACC 100.0,APO_DIST 100.0}
DECL PDAT PPDAT14={VEL 55.0,ACC 100.0,APO_DIST 100.0}
DECL PDAT PPDAT15={VEL 55.0,ACC 100.0,APO_DIST 100.0}
DECL PDAT PPDAT16={VEL 55.0,ACC 100.0,APO_DIST 100.0}
DECL E6POS XLHP090={X 1332.04504,Y -1060.80798,Z 1516.95605,A -0.00588458916,B 64.380127,C 89.9954376,S 2,T 3,E1 0.0,E2 0.0,E3 0.0,E4 0.0,E5 0.0,E6 0.0}
DECL FDAT FLHP090={TOOL_NO 1,BASE_NO 1,IPO_FRAME #BASE}
DECL PDAT PPDAT17={VEL 55.0,ACC 100.0,APO_DIST 100.0}
DECL PDAT PPDAT18={VEL 40.0,ACC 100.0,APO_DIST 100.0}
DECL PDAT PPDAT19={VEL 40.0,ACC 100.0,APO_DIST 100.0}
DECL PDAT PPDAT20={VEL 40.0,ACC 100.0,APO_DIST 100.0}
DECL PDAT PPDAT22={VEL 40.0,ACC 100.0,APO_DIST 100.0}
DECL E6POS XLHP160={X 1755.43201,Y -755.503906,Z 22.8718891,A -96.3874588,B 4.35921192,C -78.7206116,S 2,T 10,E1 0.0,E2 0.0,E3 0.0,E4 0.0,E5 0.0,E6 0.0}
DECL FDAT FLHP160={TOOL_NO 1,BASE_NO 1,IPO_FRAME #BASE}
DECL PDAT PPDAT28={VEL 100.0,ACC 100.0,APO_DIST 10.0}
DECL E6POS XLHP165={X 1586.953,Y -579.122192,Z -18.5739307,A -92.8681488,B 17.4967098,C -84.3403473,S 2,T 10,E1 0.0,E2 0.0,E3 0.0,E4 0.0,E5 0.0,E6 0.0}
DECL FDAT FLHP165={TOOL_NO 1,BASE_NO 1,IPO_FRAME #BASE}
DECL PDAT PPDAT44={VEL 100.0,ACC 100.0,APO_DIST 10.0}
DECL PDAT PPDAT45={VEL 40.0,ACC 100.0,APO_DIST 100.0}
DECL PDAT PPDAT46={VEL 40.0,ACC 100.0,APO_DIST 100.0}
DECL E6POS XLHP185={X 1558.09595,Y -603.620117,Z 12.4892702,A -87.7606506,B 11.6157598,C -89.1901627,S 2,T 10,E1 0.0,E2 0.0,E3 0.0,E4 0.0,E5 0.0,E6 0.0}
DECL FDAT FLHP185={TOOL_NO 1,BASE_NO 1,IPO_FRAME #BASE}
DECL PDAT PPDAT47={VEL 100.0,ACC 100.0,APO_DIST 100.0}
DECL PDAT PPDAT49={VEL 40.0,ACC 100.0,APO_DIST 100.0}
DECL PDAT PPDAT50={VEL 40.0,ACC 100.0,APO_DIST 100.0}
DECL PDAT PPDAT51={VEL 40.0,ACC 100.0,APO_DIST 100.0}
DECL PDAT PPDAT52={VEL 40.0,ACC 100.0,APO_DIST 100.0}
DECL E6POS XLHP200={X 1560.177,Y -438.558685,Z 136.248505,A -87.070549,B -58.6747093,C -96.842659,S 2,T 10,E1 0.0,E2 0.0,E3 0.0,E4 0.0,E5 0.0,E6 0.0}
DECL FDAT FLHP200={TOOL_NO 1,BASE_NO 1,IPO_FRAME #BASE}
DECL PDAT PPDAT53={VEL 100.0,ACC 100.0,APO_DIST 100.0}
DECL PDAT PPDAT54={VEL 40.0,ACC 100.0,APO_DIST 100.0}
DECL PDAT PPDAT55={VEL 40.0,ACC 100.0,APO_DIST 100.0}
DECL PDAT PPDAT56={VEL 55.0,ACC 100.0,APO_DIST 100.0}
DECL PDAT PPDAT57={VEL 40.0,ACC 100.0,APO_DIST 100.0}
DECL PDAT PPDAT58={VEL 55.0,ACC 100.0,APO_DIST 100.0}
DECL PDAT PPDAT59={VEL 40.0,ACC 100.0,APO_DIST 100.0}
DECL PDAT PPDAT61={VEL 40.0,ACC 100.0,APO_DIST 100.0}
DECL PDAT PPDAT62={VEL 55.0,ACC 100.0,APO_DIST 100.0}
DECL PDAT PPDAT64={VEL 40.0,ACC 100.0,APO_DIST 100.0}
DECL PDAT PPDAT65={VEL 40.0,ACC 100.0,APO_DIST 100.0}
DECL PDAT PPDAT66={VEL 40.0,ACC 100.0,APO_DIST 100.0}
DECL PDAT PPDAT67={VEL 40.0,ACC 100.0,APO_DIST 100.0}
DECL E6POS XLHP040={X 1353.50598,Y -1383.62903,Z -17.8530102,A -178.9048,B -53.4456291,C -86.9229965,S 2,T 35,E1 0.0,E2 0.0,E3 0.0,E4 0.0,E5 0.0,E6 0.0}
DECL FDAT FLHP040={TOOL_NO 1,BASE_NO 1,IPO_FRAME #BASE}
DECL PDAT PPDAT68={VEL 100.0,ACC 100.0,APO_DIST 100.0}
DECL GRP_SUGG_T LAST_GRP={NUMBER[] "1                       ",STATE[] "1                       ",PARAMS[] "GDAT0                   "}
DECL GRP_TYP GCONT={G_APO #YES,GRP_TIME 0.0,CTRL #OFF,DLY 0,DST 0}
DECL GRP_TYP GGDAT0={G_APO #NO,GRP_TIME 0.200000003,CTRL #OFF,DLY 0,DST 1}
DECL E6POS XLHP045={X 1130.30005,Y -1356.91101,Z 687.231079,A -0.546162188,B -61.9365387,C 95.6028595,S 2,T 35,E1 0.0,E2 0.0,E3 0.0,E4 0.0,E5 0.0,E6 0.0}
DECL FDAT FLHP045={TOOL_NO 1,BASE_NO 1,IPO_FRAME #BASE}
DECL PDAT PPDAT72={VEL 100.0,ACC 100.0,APO_DIST 0.0}
DECL E6POS XSWP_60_5627={X 702.076599,Y -1090.06104,Z 1422.83301,A -1.44667196,B -86.7982788,C 96.6357727,S 2,T 35,E1 0.0,E2 0.0,E3 0.0,E4 0.0,E5 0.0,E6 0.0}
DECL FDAT FSWP_60_5627={TOOL_NO 1,BASE_NO 1,IPO_FRAME #BASE}
DECL PDAT PPDAT74={VEL 50.0,ACC 100.0,APO_DIST 100.0}
DECL E6POS XSWP_60_5633={X 735.320374,Y -1090.13098,Z 1423.74597,A -1.44256198,B -86.7985916,C 96.6313477,S 2,T 35,E1 0.0,E2 0.0,E3 0.0,E4 0.0,E5 0.0,E6 0.0}
DECL FDAT FSWP_60_5633={TOOL_NO 1,BASE_NO 1,IPO_FRAME #BASE}
DECL PDAT PPDAT75={VEL 55.0,ACC 100.0,APO_DIST 100.0}
DECL E6POS XLHP055={X 749.778625,Y -1067.72803,Z 1334.35803,A -2.03584099,B -86.9460526,C 97.2368164,S 2,T 35,E1 0.0,E2 0.0,E3 0.0,E4 0.0,E5 0.0,E6 0.0}
DECL FDAT FLHP055={TOOL_NO 1,BASE_NO 1,IPO_FRAME #BASE}
DECL PDAT PPDAT76={VEL 100.0,ACC 100.0,APO_DIST 100.0}
DECL E6POS XLHP120={X 2597.70605,Y -1386.00098,Z -289.134705,A -113.716698,B 11.58113,C 0.621700227,S 2,T 3,E1 0.0,E2 0.0,E3 0.0,E4 0.0,E5 0.0,E6 0.0}
DECL FDAT FLHP120={TOOL_NO 1,BASE_NO 1,IPO_FRAME #BASE}
DECL PDAT PPDAT77={VEL 100.0,ACC 100.0,APO_DIST 100.0}
DECL E6POS XLHP030={X 1548.23303,Y -1112.33203,Z -74.4341431,A 14.8638897,B -79.8918991,C 78.3586121,S 2,T 35,E1 0.0,E2 0.0,E3 0.0,E4 0.0,E5 0.0,E6 0.0}
DECL FDAT FLHP030={TOOL_NO 1,BASE_NO 1,IPO_FRAME #BASE}
DECL PDAT PPDAT78={VEL 50.0,ACC 100.0,APO_DIST 100.0}
DECL E6POS Xp60_4371={X 1561.48804,Y -1022.66199,Z -16.1695709,A 90.1575394,B -30.7980804,C 89.7844696,S 2,T 10,E1 0.0,E2 0.0,E3 0.0,E4 0.0,E5 0.0,E6 0.0}
DECL FDAT Fp60_4371={TOOL_NO 1,BASE_NO 1,IPO_FRAME #BASE}
DECL E6POS XP60_4351={X 1558.62,Y -653.484985,Z -46.1423187,A -88.1710663,B 12.8774996,C -89.4586334,S 2,T 10,E1 0.0,E2 0.0,E3 0.0,E4 0.0,E5 0.0,E6 0.0}
DECL FDAT Fp60_4351={TOOL_NO 1,BASE_NO 1,IPO_FRAME #BASE}
DECL E6POS Xp60_4349={X 1559.17102,Y -629.641724,Z -19.6255398,A -88.0318909,B 11.5881004,C -92.0015564,S 2,T 10,E1 0.0,E2 0.0,E3 0.0,E4 0.0,E5 0.0,E6 0.0}
DECL FDAT Fp60_4349={TOOL_NO 1,BASE_NO 1,IPO_FRAME #BASE}
DECL E6POS Xp60_4343={X 1560.55798,Y -605.862488,Z 85.4798737,A -89.4882507,B 1.53147805,C -89.0940094,S 2,T 10,E1 0.0,E2 0.0,E3 0.0,E4 0.0,E5 0.0,E6 0.0}
DECL FDAT Fp60_4343={TOOL_NO 1,BASE_NO 1,IPO_FRAME #BASE}
DECL E6POS Xp60_4337={X 1564.27698,Y -509.893799,Z 160.744202,A -92.2010269,B 1.71480799,C -92.1405869,S 2,T 10,E1 0.0,E2 0.0,E3 0.0,E4 0.0,E5 0.0,E6 0.0}
DECL FDAT Fp60_4337={TOOL_NO 1,BASE_NO 1,IPO_FRAME #BASE}
DECL E6POS Xp60_4339={X 1562.60205,Y -542.482727,Z 141.984497,A -91.9770432,B 1.58319402,C -91.9299011,S 2,T 10,E1 0.0,E2 0.0,E3 0.0,E4 0.0,E5 0.0,E6 0.0}
DECL FDAT Fp60_4339={TOOL_NO 1,BASE_NO 1,IPO_FRAME #BASE}
DECL E6POS XLHP195={X 1561.172,Y -483.440399,Z 112.178802,A -91.7479172,B -10.31639,C -92.1747437,S 2,T 10,E1 0.0,E2 0.0,E3 0.0,E4 0.0,E5 0.0,E6 0.0}
DECL FDAT FLHP195={TOOL_NO 1,BASE_NO 1,IPO_FRAME #BASE}
DECL PDAT PPDAT81={VEL 100.0,ACC 100.0,APO_DIST 100.0}
DECL E6POS Xp60_4333={X 1565.56604,Y -462.748505,Z 209.144196,A -90.4667435,B -49.8350792,C -93.3813934,S 2,T 10,E1 0.0,E2 0.0,E3 0.0,E4 0.0,E5 0.0,E6 0.0}
DECL FDAT Fp60_4333={TOOL_NO 1,BASE_NO 1,IPO_FRAME #BASE}
DECL E6POS Xp60_4331={X 1565.97803,Y -444.523102,Z 241.732697,A -90.4668732,B -49.8349991,C -93.3811188,S 2,T 10,E1 0.0,E2 0.0,E3 0.0,E4 0.0,E5 0.0,E6 0.0}
DECL FDAT Fp60_4331={TOOL_NO 1,BASE_NO 1,IPO_FRAME #BASE}
DECL E6POS XLHP205={X 1565.771,Y -403.419495,Z 266.34729,A -85.9189987,B -72.9562836,C -97.4569321,S 2,T 10,E1 0.0,E2 0.0,E3 0.0,E4 0.0,E5 0.0,E6 0.0}
DECL FDAT FLHP205={TOOL_NO 1,BASE_NO 1,IPO_FRAME #BASE}
DECL PDAT PPDAT82={VEL 100.0,ACC 100.0,APO_DIST 100.0}
DECL E6POS XP60_4327={X 1568.125,Y -407.928986,Z 303.251312,A -85.9195099,B -72.956131,C -97.4564972,S 2,T 10,E1 0.0,E2 0.0,E3 0.0,E4 0.0,E5 0.0,E6 0.0}
DECL FDAT Fp60_4327={TOOL_NO 1,BASE_NO 1,IPO_FRAME #BASE}
DECL E6POS XP60_4325={X 1567.43506,Y -387.418701,Z 322.787415,A -85.9231033,B -72.9556808,C -97.4537888,S 2,T 10,E1 0.0,E2 0.0,E3 0.0,E4 0.0,E5 0.0,E6 0.0}
DECL FDAT Fp60_4325={TOOL_NO 1,BASE_NO 1,IPO_FRAME #BASE}
DECL E6POS XLHP210={X 1563.34595,Y -349.733612,Z 318.417206,A -71.4139023,B -84.1100464,C -111.742699,S 2,T 10,E1 0.0,E2 0.0,E3 0.0,E4 0.0,E5 0.0,E6 0.0}
DECL FDAT FLHP210={TOOL_NO 1,BASE_NO 1,IPO_FRAME #BASE}
DECL PDAT PPDAT83={VEL 100.0,ACC 100.0,APO_DIST 100.0}
DECL E6POS XP60_4321={X 1567.80396,Y -334.62381,Z 351.912994,A -71.4166794,B -84.1095581,C -111.739998,S 2,T 10,E1 0.0,E2 0.0,E3 0.0,E4 0.0,E5 0.0,E6 0.0}
DECL FDAT Fp60_4321={TOOL_NO 1,BASE_NO 1,IPO_FRAME #BASE}
DECL E6POS XP60_4319={X 1568.41199,Y -307.219208,Z 357.307709,A -71.4183502,B -84.1091766,C -111.738503,S 2,T 10,E1 0.0,E2 0.0,E3 0.0,E4 0.0,E5 0.0,E6 0.0}
DECL FDAT Fp60_4319={TOOL_NO 1,BASE_NO 1,IPO_FRAME #BASE}
DECL E6POS XP60_4315={X 1567.14001,Y -251.587494,Z 359.020111,A -71.418869,B -84.110321,C -111.738197,S 2,T 10,E1 0.0,E2 0.0,E3 0.0,E4 0.0,E5 0.0,E6 0.0}
DECL FDAT Fp60_4315={TOOL_NO 1,BASE_NO 1,IPO_FRAME #BASE}
DECL PDAT PPDAT84={VEL 40.0,ACC 100.0,APO_DIST 100.0}
DECL E6POS XP60_4313={X 1566.75195,Y -220.066101,Z 358.25769,A -71.4223175,B -84.1103516,C -111.7342,S 2,T 10,E1 0.0,E2 0.0,E3 0.0,E4 0.0,E5 0.0,E6 0.0}
DECL FDAT Fp60_4313={TOOL_NO 1,BASE_NO 1,IPO_FRAME #BASE}
DECL E6POS XLHP215={X 1564.93506,Y -189.126694,Z 322.113098,A 83.0863571,B -60.54739,C 94.4320831,S 2,T 10,E1 0.0,E2 0.0,E3 0.0,E4 0.0,E5 0.0,E6 0.0}
DECL FDAT FLHP215={TOOL_NO 1,BASE_NO 1,IPO_FRAME #BASE}
DECL PDAT PPDAT85={VEL 100.0,ACC 100.0,APO_DIST 100.0}
DECL E6POS XP60_4309={X 1566.28198,Y -161.240204,Z 360.502594,A 83.0860367,B -60.5472298,C 94.4322433,S 2,T 10,E1 0.0,E2 0.0,E3 0.0,E4 0.0,E5 0.0,E6 0.0}
DECL FDAT Fp60_4309={TOOL_NO 1,BASE_NO 1,IPO_FRAME #BASE}
DECL E6POS XP60_4305={X 1566.01599,Y -97.0816193,Z 360.544312,A 83.0888367,B -60.5480003,C 94.4286499,S 2,T 10,E1 0.0,E2 0.0,E3 0.0,E4 0.0,E5 0.0,E6 0.0}
DECL FDAT Fp60_4305={TOOL_NO 1,BASE_NO 1,IPO_FRAME #BASE}
DECL E6POS XP60_4303={X 1564.64502,Y -65.7111969,Z 360.644897,A 83.086937,B -60.5485001,C 94.4319305,S 2,T 10,E1 0.0,E2 0.0,E3 0.0,E4 0.0,E5 0.0,E6 0.0}
DECL FDAT Fp60_4303={TOOL_NO 1,BASE_NO 1,IPO_FRAME #BASE}
DECL E6POS XP60_4301={X 1564.98303,Y -31.4840603,Z 359.913788,A 83.0870819,B -60.5491905,C 94.431778,S 2,T 10,E1 0.0,E2 0.0,E3 0.0,E4 0.0,E5 0.0,E6 0.0}
DECL FDAT Fp60_4301={TOOL_NO 1,BASE_NO 1,IPO_FRAME #BASE}
DECL E6POS XP60_4300={X 1565.14502,Y -1.88436699,Z 359.564697,A 83.0881424,B -60.5521011,C 94.4303284,S 2,T 10,E1 0.0,E2 0.0,E3 0.0,E4 0.0,E5 0.0,E6 0.0}
DECL FDAT Fp60_4300={TOOL_NO 1,BASE_NO 1,IPO_FRAME #BASE}
DECL E6POS XLHP170={X 2324.63599,Y 1443.38794,Z 998.726501,A -179.109497,B 4.75907278,C -85.1163101,S 2,T 10,E1 0.0,E2 0.0,E3 0.0,E4 0.0,E5 0.0,E6 0.0}
DECL FDAT FLHP170={TOOL_NO 1,BASE_NO 0,IPO_FRAME #BASE}
DECL PDAT PPDAT86={VEL 100.0,ACC 100.0,APO_DIST 10.0}
DECL E6POS XLHP175={X 2206.53809,Y 1431.41895,Z 996.117676,A -178.806198,B -1.14055502,C -86.5652618,S 2,T 10,E1 0.0,E2 0.0,E3 0.0,E4 0.0,E5 0.0,E6 0.0}
DECL FDAT FLHP175={TOOL_NO 1,BASE_NO 0,IPO_FRAME #BASE}
DECL PDAT PPDAT87={VEL 100.0,ACC 100.0,APO_DIST 5.0}
DECL E6POS XLHP180={X 2177.60107,Y 1429.94104,Z 1005.08502,A -179.462997,B -11.9197798,C -86.49086,S 2,T 10,E1 0.0,E2 0.0,E3 0.0,E4 0.0,E5 0.0,E6 0.0}
DECL FDAT FLHP180={TOOL_NO 1,BASE_NO 0,IPO_FRAME #BASE}
DECL PDAT PPDAT88={VEL 100.0,ACC 100.0,APO_DIST 100.0}
DECL E6POS XSWP_60_4357={X 1558.17395,Y -756.874329,Z -56.0067902,A -89.4890137,B -12.1817703,C -87.7156372,S 2,T 10,E1 0.0,E2 0.0,E3 0.0,E4 0.0,E5 0.0,E6 0.0}
DECL FDAT Fswp_60_4357={TOOL_NO 1,BASE_NO 1,IPO_FRAME #BASE}
DECL PDAT PPDAT89={VEL 40.0,ACC 100.0,APO_DIST 100.0}
DECL E6POS XSWP_60_4355={X 1559.80005,Y -719.43811,Z -55.1353607,A -89.5820313,B -12.2156,C -88.8096085,S 2,T 10,E1 0.0,E2 0.0,E3 0.0,E4 0.0,E5 0.0,E6 0.0}
DECL FDAT Fswp_60_4355={TOOL_NO 1,BASE_NO 1,IPO_FRAME #BASE}
DECL PDAT PPDAT90={VEL 40.0,ACC 100.0,APO_DIST 100.0}
DECL E6POS Xswp_60_4413={X 1488.16797,Y -1114.09705,Z -20.2259102,A 173.440002,B -78.3635864,C -79.8442001,S 2,T 35,E1 0.0,E2 0.0,E3 0.0,E4 0.0,E5 0.0,E6 0.0}
DECL FDAT Fswp_60_4413={TOOL_NO 1,BASE_NO 1,IPO_FRAME #BASE}
DECL E6POS Xswp_60_4405={X 1512.66199,Y -1112.65796,Z -21.0145302,A 173.438904,B -78.3632813,C -79.8431931,S 2,T 35,E1 0.0,E2 0.0,E3 0.0,E4 0.0,E5 0.0,E6 0.0}
DECL FDAT Fswp_60_4405={TOOL_NO 1,BASE_NO 1,IPO_FRAME #BASE}
DECL E6POS Xswp_60_4409={X 1546.90198,Y -1110.72095,Z -21.4948997,A 161.011002,B -84.6591187,C -67.5320129,S 2,T 35,E1 0.0,E2 0.0,E3 0.0,E4 0.0,E5 0.0,E6 0.0}
DECL FDAT Fswp_60_4409={TOOL_NO 1,BASE_NO 1,IPO_FRAME #BASE}
DECL E6POS Xswp_60_4663={X 1323.11499,Y -1061.59399,Z 1508.94202,A -0.00694822101,B 64.3793106,C 89.9941711,S 2,T 3,E1 0.0,E2 0.0,E3 0.0,E4 0.0,E5 0.0,E6 0.0}
DECL FDAT Fswp_60_4663={TOOL_NO 1,BASE_NO 1,IPO_FRAME #BASE}
DECL E6POS Xswp_60_4667={X 1322.64197,Y -1061.48303,Z 1480.97498,A -0.00707656285,B 64.3793335,C 89.9941864,S 2,T 3,E1 0.0,E2 0.0,E3 0.0,E4 0.0,E5 0.0,E6 0.0}
DECL FDAT Fswp_60_4667={TOOL_NO 1,BASE_NO 1,IPO_FRAME #BASE}
DECL E6POS Xswp_60_4671={X 1321.198,Y -1061.80896,Z 1452.18701,A -0.00710433302,B 64.3792801,C 89.9941025,S 2,T 3,E1 0.0,E2 0.0,E3 0.0,E4 0.0,E5 0.0,E6 0.0}
DECL FDAT Fswp_60_4671={TOOL_NO 1,BASE_NO 1,IPO_FRAME #BASE}
DECL E6POS Xswp_60_4675={X 1349.94104,Y -1060.61804,Z 1452.60596,A -0.00707376003,B 64.3794632,C 89.9942093,S 2,T 3,E1 0.0,E2 0.0,E3 0.0,E4 0.0,E5 0.0,E6 0.0}
DECL FDAT Fswp_60_4675={TOOL_NO 1,BASE_NO 1,IPO_FRAME #BASE}
DECL E6POS Xswp_60_4669={X 1350.83301,Y -1060.93701,Z 1480.29395,A -0.006768052,B 64.3794937,C 89.9944534,S 2,T 3,E1 0.0,E2 0.0,E3 0.0,E4 0.0,E5 0.0,E6 0.0}
DECL FDAT Fswp_60_4669={TOOL_NO 1,BASE_NO 1,IPO_FRAME #BASE}
DECL E6POS Xswp_60_4665={X 1352.48596,Y -1060.43799,Z 1508.38403,A -0.00652889023,B 64.3795929,C 89.9946671,S 2,T 3,E1 0.0,E2 0.0,E3 0.0,E4 0.0,E5 0.0,E6 0.0}
DECL FDAT Fswp_60_4665={TOOL_NO 1,BASE_NO 1,IPO_FRAME #BASE}
DECL E6POS Xswp_60_4369={X 1561.90906,Y -990.627808,Z -16.3027,A 90.0004425,B -27.9580498,C 89.9998016,S 2,T 10,E1 0.0,E2 0.0,E3 0.0,E4 0.0,E5 0.0,E6 0.0}
DECL FDAT Fswp_60_4369={TOOL_NO 1,BASE_NO 1,IPO_FRAME #BASE}
DECL E6POS Xswp_60_4365={X 1562.10498,Y -916.611023,Z -25.0478592,A 90.0004501,B -16.1103191,C 89.9994812,S 2,T 10,E1 0.0,E2 0.0,E3 0.0,E4 0.0,E5 0.0,E6 0.0}
DECL FDAT Fswp_60_4365={TOOL_NO 1,BASE_NO 1,IPO_FRAME #BASE}
DECL E6POS Xswp_60_4361={X 1559.65503,Y -878.630676,Z -34.7861404,A 90.0006714,B -10.9229803,C 89.9998169,S 2,T 10,E1 0.0,E2 0.0,E3 0.0,E4 0.0,E5 0.0,E6 0.0}
DECL FDAT Fswp_60_4361={TOOL_NO 1,BASE_NO 1,IPO_FRAME #BASE}
DECL E6POS Xswp_60_4345={X 1561.62598,Y -615.966125,Z 49.6089897,A -84.9490967,B -2.45235705,C -91.1025314,S 2,T 10,E1 0.0,E2 0.0,E3 0.0,E4 0.0,E5 0.0,E6 0.0}
DECL FDAT Fswp_60_4345={TOOL_NO 1,BASE_NO 1,IPO_FRAME #BASE}
DECL E6POS XLHP240={X 2562.45093,Y -1774.07495,Z -228.403,A -159.798798,B -5.811625,C -4.77948093,S 2,T 10,E1 0.0,E2 0.0,E3 0.0,E4 0.0,E5 0.0,E6 0.0}
DECL FDAT FLHP240={TOOL_NO 1,BASE_NO 1,IPO_FRAME #BASE}
DECL PDAT PPDAT91={VEL 100.0,ACC 100.0,APO_DIST 100.0}
DECL E6POS XP60_4307={X 1567.56006,Y -129.819702,Z 360.834198,A 83.0858917,B -60.5472488,C 94.4323273,S 2,T 10,E1 0.0,E2 0.0,E3 0.0,E4 0.0,E5 0.0,E6 0.0}
DECL FDAT Fp60_4307={TOOL_NO 1,BASE_NO 1,IPO_FRAME #BASE}
DECL PDAT PPDAT92={VEL 40.0,ACC 100.0,APO_DIST 100.0}
DECL E6POS XLHP050={X 706.573914,Y -1090.27197,Z 1335.42102,A -2.03537107,B -86.945343,C 97.2361832,S 2,T 35,E1 0.0,E2 0.0,E3 0.0,E4 0.0,E5 0.0,E6 0.0}
DECL FDAT FLHP050={TOOL_NO 1,BASE_NO 1,IPO_FRAME #BASE}
DECL PDAT PPDAT93={VEL 100.0,ACC 100.0,APO_DIST 10.0}
DECL E6POS XLHP005={X 1013.06097,Y -2516.00391,Z 240.248001,A 90.0,B 0.0,C 34.9999008,S 2,T 43}
DECL FDAT FLHP005={TOOL_NO 1,BASE_NO 1,IPO_FRAME #BASE}
DECL BASIS_SUGG_T LAST_BASIS={POINT1[] "PS01010001              ",POINT2[] "PS01010001              ",CP_PARAMS[] "CPDAT0                  ",PTP_PARAMS[] "PDAT0                   ",CONT[] "                        ",CP_VEL[] "2.0                     ",PTP_VEL[] " 100                    ",SPL_NAME[] "S0                      "}
ENDDAT
